METHOD TryMakeReferenceTo : BOOL
VAR_INPUT
	Target : I_Datatype;
END_VAR
VAR
	pTargetData : POINTER TO ETcVnOcrModelType;
END_VAR
IF NOT IsEquivalentTo(Target) THEN
	RETURN;
END_IF

pTargetData := Target.Address;
activeData REF= pTargetData^;
SetBaseDatatypeReference();
TryMakeReferenceTo := TRUE;
END_METHOD

PROPERTY PUBLIC Value : ETcVnOcrModelType
GET
Value := activeData;
END_GET
SET
activeData := Value;
END_SET
END_PROPERTY

END_FUNCTION_BLOCK

// ---- Datatypes/Enums/_ETcVnTimestamp.TcPOU
{attribute 'linkalways'} 
{attribute 'no_explicit_call' := 'This FB is a CLASS and must be accessed using methods or properties'}
{attribute 'enable_dynamic_creation'}
FUNCTION_BLOCK _ETcVnTimestamp EXTENDS EnumDatatypeBase
VAR
	localData : ETcVnTimestamp;
	activeData : REFERENCE TO ETcVnTimestamp;
	enumBaseDatatype : _ULINT(localData);
END_VAR

METHOD PRIVATE AddLocalEnumeration
VAR_INPUT
	Enumeration : T_MAXSTRING;
	Value : ETcVnTimestamp;
END_VAR
AddEnumeration(Enumeration, Value);
END_METHOD

PROPERTY PUBLIC Address : PVOID
GET
Address := ADR(activeData);
END_GET
END_PROPERTY

METHOD PUBLIC ClearReference
VAR_INPUT
END_VAR
activeData REF= localData;
SetBaseDatatypeReference();
END_METHOD

METHOD PUBLIC Clone : I_Datatype
VAR
    pClone : POINTER TO _ETcVnTimestamp;
END_VAR
pClone := __NEW(_ETcVnTimestamp(InitialValue := Value));
Clone := pClone^;
END_METHOD

METHOD FB_init : BOOL
VAR_INPUT
	bInitRetains : BOOL; // if TRUE, the retain variables are initialized (warm start / cold start)
	bInCopyCode : BOOL;  // if TRUE, the instance afterwards gets moved into the copy code (online change)
	InitialValue : ETcVnTimestamp;
END_VAR
localData := InitialValue;
AddBaseDatatype(enumBaseDatatype);
ClearReference();

AddLocalEnumeration('TCVN_TS_IMAGE_COMPLETED', ETcVnTimestamp.TCVN_TS_IMAGE_COMPLETED);
END_METHOD

PROPERTY PUBLIC Identifier : T_MAXSTRING
GET
Identifier := 'ETcVnTimestamp';
END_GET
END_PROPERTY

METHOD IsEnumeratorValueEqual : BOOL
VAR_INPUT
	Enumerator : I_KeyValueForwardEnumerator;
END_VAR
VAR
	storedValue : ETcVnTimestamp;
END_VAR
IF NOT Enumerator.TryGet(storedValue) THEN
	RETURN;
END_IF

IsEnumeratorValueEqual := storedValue = activeData;
END_METHOD

METHOD PUBLIC MakeReferenceTo
VAR_INPUT
	ReferenceTarget : REFERENCE TO ETcVnTimestamp;
END_VAR
activeData REF= ReferenceTarget;
SetBaseDatatypeReference();
END_METHOD

METHOD PROTECTED SetBaseDatatypeReference
VAR_INPUT
END_VAR
enumBaseDatatype.MakeReferenceTo(activeData);
END_METHOD

PROPERTY PUBLIC Size : UDINT
GET
Size := SIZEOF(activeData);
END_GET
END_PROPERTY

METHOD TryMakeReferenceTo : BOOL
VAR_INPUT
	Target : I_Datatype;
END_VAR
VAR
	pTargetData : POINTER TO ETcVnTimestamp;
END_VAR
IF NOT IsEquivalentTo(Target) THEN
	RETURN;
END_IF

pTargetData := Target.Address;
activeData REF= pTargetData^;
SetBaseDatatypeReference();
TryMakeReferenceTo := TRUE;
END_METHOD

PROPERTY PUBLIC Value : ETcVnTimestamp
GET
Value := activeData;
END_GET
SET
activeData := Value;
END_SET
END_PROPERTY

END_FUNCTION_BLOCK

// ---- Datatypes/Enums/_ETcVnOcrOptions.TcPOU
{attribute 'linkalways'} 
{attribute 'no_explicit_call' := 'This FB is a CLASS and must be accessed using methods or properties'}
{attribute 'enable_dynamic_creation'}
FUNCTION_BLOCK _ETcVnOcrOptions EXTENDS EnumDatatypeBase
VAR
	localData : ETcVnOcrOptions;
	activeData : REFERENCE TO ETcVnOcrOptions;
	enumBaseDatatype : _UDINT(localData);
END_VAR

METHOD PRIVATE AddLocalEnumeration
VAR_INPUT
	Enumeration : T_MAXSTRING;
	Value : ETcVnOcrOptions;
END_VAR
AddEnumeration(Enumeration, Value);
END_METHOD

PROPERTY PUBLIC Address : PVOID
GET
Address := ADR(activeData);
END_GET
END_PROPERTY

METHOD PUBLIC ClearReference
VAR_INPUT
END_VAR
activeData REF= localData;
SetBaseDatatypeReference();
END_METHOD

METHOD PUBLIC Clone : I_Datatype
VAR
    pClone : POINTER TO _ETcVnOcrOptions;
END_VAR
pClone := __NEW(_ETcVnOcrOptions(InitialValue := Value));
Clone := pClone^;
END_METHOD

METHOD FB_init : BOOL
VAR_INPUT
	bInitRetains : BOOL; // if TRUE, the retain variables are initialized (warm start / cold start)
	bInCopyCode : BOOL;  // if TRUE, the instance afterwards gets moved into the copy code (online change)
	InitialValue : ETcVnOcrOptions;
END_VAR
localData := InitialValue;
AddBaseDatatype(enumBaseDatatype);
ClearReference();

AddLocalEnumeration('TCVN_OO_WITHBLANKS', ETcVnOcrOptions.TCVN_OO_WITHBLANKS);
END_METHOD

PROPERTY PUBLIC Identifier : T_MAXSTRING
GET
Identifier := 'ETcVnOcrOptions';
END_GET
END_PROPERTY

METHOD IsEnumeratorValueEqual : BOOL
VAR_INPUT
	Enumerator : I_KeyValueForwardEnumerator;
END_VAR
VAR
	storedValue : ETcVnOcrOptions;
END_VAR
IF NOT Enumerator.TryGet(storedValue) THEN
	RETURN;
END_IF

IsEnumeratorValueEqual := storedValue = activeData;
END_METHOD

METHOD PUBLIC MakeReferenceTo
VAR_INPUT
	ReferenceTarget : REFERENCE TO ETcVnOcrOptions;
END_VAR
activeData REF= ReferenceTarget;
SetBaseDatatypeReference();
END_METHOD

METHOD PROTECTED SetBaseDatatypeReference
VAR_INPUT
END_VAR
enumBaseDatatype.MakeReferenceTo(activeData);
END_METHOD

PROPERTY PUBLIC Size : UDINT
GET
Size := SIZEOF(activeData);
END_GET
END_PROPERTY

METHOD TryMakeReferenceTo : BOOL
VAR_INPUT
	Target : I_Datatype;
END_VAR
VAR
	pTargetData : POINTER TO ETcVnOcrOptions;
END_VAR
IF NOT IsEquivalentTo(Target) THEN
	RETURN;
END_IF

pTargetData := Target.Address;
activeData REF= pTargetData^;
SetBaseDatatypeReference();
TryMakeReferenceTo := TRUE;
END_METHOD

PROPERTY PUBLIC Value : ETcVnOcrOptions
GET
Value := activeData;
END_GET
SET
activeData := Value;
END_SET
END_PROPERTY

END_FUNCTION_BLOCK

// ---- Datatypes/Enums/_ETcVnOrientationMethod.TcPOU
{attribute 'linkalways'} 
{attribute 'no_explicit_call' := 'This FB is a CLASS and must be accessed using methods or properties'}
{attribute 'enable_dynamic_creation'}
FUNCTION_BLOCK _ETcVnOrientationMethod EXTENDS EnumDatatypeBase
VAR
	localData : ETcVnOrientationMethod;
	activeData : REFERENCE TO ETcVnOrientationMethod;
	enumBaseDatatype : _DINT(localData);
END_VAR

METHOD PRIVATE AddLocalEnumeration
VAR_INPUT
	Enumeration : T_MAXSTRING;
	Value : ETcVnOrientationMethod;
END_VAR
AddEnumeration(Enumeration, Value);
END_METHOD

PROPERTY PUBLIC Address : PVOID
GET
Address := ADR(activeData);
END_GET
END_PROPERTY

METHOD PUBLIC ClearReference
VAR_INPUT
END_VAR
activeData REF= localData;
SetBaseDatatypeReference();
END_METHOD

METHOD PUBLIC Clone : I_Datatype
VAR
    pClone : POINTER TO _ETcVnOrientationMethod;
END_VAR
pClone := __NEW(_ETcVnOrientationMethod(InitialValue := Value));
Clone := pClone^;
END_METHOD

METHOD FB_init : BOOL
VAR_INPUT
	bInitRetains : BOOL; // if TRUE, the retain variables are initialized (warm start / cold start)
	bInCopyCode : BOOL;  // if TRUE, the instance afterwards gets moved into the copy code (online change)
	InitialValue : ETcVnOrientationMethod;
END_VAR
localData := InitialValue;
AddBaseDatatype(enumBaseDatatype);
ClearReference();

AddLocalEnumeration('TCVN_OM_PCA', ETcVnOrientationMethod.TCVN_OM_PCA);
AddLocalEnumeration('TCVN_OM_FITELLIPSE', ETcVnOrientationMethod.TCVN_OM_FITELLIPSE);
AddLocalEnumeration('TCVN_OM_MOMENTS', ETcVnOrientationMethod.TCVN_OM_MOMENTS);
AddLocalEnumeration('TCVN_OM_ENCLOSINGRECT', ETcVnOrientationMethod.TCVN_OM_ENCLOSINGRECT);
END_METHOD

PROPERTY PUBLIC Identifier : T_MAXSTRING
GET
Identifier := 'ETcVnOrientationMethod';
END_GET
END_PROPERTY

METHOD IsEnumeratorValueEqual : BOOL
VAR_INPUT
	Enumerator : I_KeyValueForwardEnumerator;
END_VAR
VAR
	storedValue : ETcVnOrientationMethod;
END_VAR
IF NOT Enumerator.TryGet(storedValue) THEN
	RETURN;
END_IF

IsEnumeratorValueEqual := storedValue = activeData;
END_METHOD

METHOD PUBLIC MakeReferenceTo
VAR_INPUT
	ReferenceTarget : REFERENCE TO ETcVnOrientationMethod;
END_VAR
activeData REF= ReferenceTarget;
SetBaseDatatypeReference();
END_METHOD

METHOD PROTECTED SetBaseDatatypeReference
VAR_INPUT
END_VAR
enumBaseDatatype.MakeReferenceTo(activeData);
END_METHOD

PROPERTY PUBLIC Size : UDINT
GET
Size := SIZEOF(activeData);
END_GET
END_PROPERTY

METHOD TryMakeReferenceTo : BOOL
VAR_INPUT
	Target : I_Datatype;
END_VAR
VAR
	pTargetData : POINTER TO ETcVnOrientationMethod;
END_VAR
IF NOT IsEquivalentTo(Target) THEN
	RETURN;
END_IF

pTargetData := Target.Address;
activeData REF= pTargetData^;
SetBaseDatatypeReference();
TryMakeReferenceTo := TRUE;
END_METHOD

PROPERTY PUBLIC Value : ETcVnOrientationMethod
GET
Value := activeData;
END_GET
SET
activeData := Value;
END_SET
END_PROPERTY

END_FUNCTION_BLOCK

// ---- Datatypes/Enums/_ETcVnPaddingMode.TcPOU
{attribute 'linkalways'} 
{attribute 'no_explicit_call' := 'This FB is a CLASS and must be accessed using methods or properties'}
{attribute 'enable_dynamic_creation'}
FUNCTION_BLOCK _ETcVnPaddingMode EXTENDS EnumDatatypeBase
VAR
	localData : ETcVnPaddingMode;
	activeData : REFERENCE TO ETcVnPaddingMode;
	enumBaseDatatype : _DINT(localData);
END_VAR

METHOD PRIVATE AddLocalEnumeration
VAR_INPUT
	Enumeration : T_MAXSTRING;
	Value : ETcVnPaddingMode;
END_VAR
AddEnumeration(Enumeration, Value);
END_METHOD

PROPERTY PUBLIC Address : PVOID
GET
Address := ADR(activeData);
END_GET
END_PROPERTY

METHOD PUBLIC ClearReference
VAR_INPUT
END_VAR
activeData REF= localData;
SetBaseDatatypeReference();
END_METHOD

METHOD PUBLIC Clone : I_Datatype
VAR
    pClone : POINTER TO _ETcVnPaddingMode;
END_VAR
pClone := __NEW(_ETcVnPaddingMode(InitialValue := Value));
Clone := pClone^;
END_METHOD

METHOD FB_init : BOOL
VAR_INPUT
	bInitRetains : BOOL; // if TRUE, the retain variables are initialized (warm start / cold start)
	bInCopyCode : BOOL;  // if TRUE, the instance afterwards gets moved into the copy code (online change)
	InitialValue : ETcVnPaddingMode;
END_VAR
localData := InitialValue;
AddBaseDatatype(enumBaseDatatype);
ClearReference();

AddLocalEnumeration('TCVN_PM_NONE', ETcVnPaddingMode.TCVN_PM_NONE);
AddLocalEnumeration('TCVN_PM_CROP_CENTER', ETcVnPaddingMode.TCVN_PM_CROP_CENTER);
AddLocalEnumeration('TCVN_PM_LETTERBOX', ETcVnPaddingMode.TCVN_PM_LETTERBOX);
END_METHOD

PROPERTY PUBLIC Identifier : T_MAXSTRING
GET
Identifier := 'ETcVnPaddingMode';
END_GET
END_PROPERTY

METHOD IsEnumeratorValueEqual : BOOL
VAR_INPUT
	Enumerator : I_KeyValueForwardEnumerator;
END_VAR
VAR
	storedValue : ETcVnPaddingMode;
END_VAR
IF NOT Enumerator.TryGet(storedValue) THEN
	RETURN;
END_IF

IsEnumeratorValueEqual := storedValue = activeData;
END_METHOD

METHOD PUBLIC MakeReferenceTo
VAR_INPUT
	ReferenceTarget : REFERENCE TO ETcVnPaddingMode;
END_VAR
activeData REF= ReferenceTarget;
SetBaseDatatypeReference();
END_METHOD

METHOD PROTECTED SetBaseDatatypeReference
VAR_INPUT
END_VAR
enumBaseDatatype.MakeReferenceTo(activeData);
END_METHOD

PROPERTY PUBLIC Size : UDINT
GET
Size := SIZEOF(activeData);
END_GET
END_PROPERTY

METHOD TryMakeReferenceTo : BOOL
VAR_INPUT
	Target : I_Datatype;
END_VAR
VAR
	pTargetData : POINTER TO ETcVnPaddingMode;
END_VAR
IF NOT IsEquivalentTo(Target) THEN
	RETURN;
END_IF

pTargetData := Target.Address;
activeData REF= pTargetData^;
SetBaseDatatypeReference();
TryMakeReferenceTo := TRUE;
END_METHOD

PROPERTY PUBLIC Value : ETcVnPaddingMode
GET
Value := activeData;
END_GET
SET
activeData := Value;
END_SET
END_PROPERTY

END_FUNCTION_BLOCK

// ---- Datatypes/Enums/_ETcVnPixelConnectivity.TcPOU
{attribute 'linkalways'} 
{attribute 'no_explicit_call' := 'This FB is a CLASS and must be accessed using methods or properties'}
{attribute 'enable_dynamic_creation'}
FUNCTION_BLOCK _ETcVnPixelConnectivity EXTENDS EnumDatatypeBase
VAR
	localData : ETcVnPixelConnectivity;
	activeData : REFERENCE TO ETcVnPixelConnectivity;
	enumBaseDatatype : _DINT(localData);
END_VAR

METHOD PRIVATE AddLocalEnumeration
VAR_INPUT
	Enumeration : T_MAXSTRING;
	Value : ETcVnPixelConnectivity;
END_VAR
AddEnumeration(Enumeration, Value);
END_METHOD

PROPERTY PUBLIC Address : PVOID
GET
Address := ADR(activeData);
END_GET
END_PROPERTY

METHOD PUBLIC ClearReference
VAR_INPUT
END_VAR
activeData REF= localData;
SetBaseDatatypeReference();
END_METHOD

METHOD PUBLIC Clone : I_Datatype
VAR
    pClone : POINTER TO _ETcVnPixelConnectivity;
END_VAR
pClone := __NEW(_ETcVnPixelConnectivity(InitialValue := Value));
Clone := pClone^;
END_METHOD

METHOD FB_init : BOOL
VAR_INPUT
	bInitRetains : BOOL; // if TRUE, the retain variables are initialized (warm start / cold start)
	bInCopyCode : BOOL;  // if TRUE, the instance afterwards gets moved into the copy code (online change)
	InitialValue : ETcVnPixelConnectivity;
END_VAR
localData := InitialValue;
AddBaseDatatype(enumBaseDatatype);
ClearReference();

AddLocalEnumeration('TCVN_PC_4', ETcVnPixelConnectivity.TCVN_PC_4);
AddLocalEnumeration('TCVN_PC_8', ETcVnPixelConnectivity.TCVN_PC_8);
END_METHOD

PROPERTY PUBLIC Identifier : T_MAXSTRING
GET
Identifier := 'ETcVnPixelConnectivity';
END_GET
END_PROPERTY

METHOD IsEnumeratorValueEqual : BOOL
VAR_INPUT
	Enumerator : I_KeyValueForwardEnumerator;
END_VAR
VAR
	storedValue : ETcVnPixelConnectivity;
END_VAR
IF NOT Enumerator.TryGet(storedValue) THEN
	RETURN;
END_IF

IsEnumeratorValueEqual := storedValue = activeData;
END_METHOD

METHOD PUBLIC MakeReferenceTo
VAR_INPUT
	ReferenceTarget : REFERENCE TO ETcVnPixelConnectivity;
END_VAR
activeData REF= ReferenceTarget;
SetBaseDatatypeReference();
END_METHOD

METHOD PROTECTED SetBaseDatatypeReference
VAR_INPUT
END_VAR
enumBaseDatatype.MakeReferenceTo(activeData);
END_METHOD

PROPERTY PUBLIC Size : UDINT
GET
Size := SIZEOF(activeData);
END_GET
END_PROPERTY

METHOD TryMakeReferenceTo : BOOL
VAR_INPUT
	Target : I_Datatype;
END_VAR
VAR
	targetAsEnum : I_EnumDatatype;
	pTargetData : POINTER TO ETcVnPixelConnectivity;
END_VAR
IF NOT Target.TryResolveAsEnumDatatype(targetAsEnum) THEN
	RETURN;
END_IF

IF targetAsEnum.Identifier <> Identifier THEN
	RETURN;
END_IF

pTargetData := Target.Address;
activeData REF= pTargetData^;
SetBaseDatatypeReference();
TryMakeReferenceTo := TRUE;
END_METHOD

PROPERTY PUBLIC Value : ETcVnPixelConnectivity
GET
Value := activeData;
END_GET
SET
activeData := Value;
END_SET
END_PROPERTY

END_FUNCTION_BLOCK

// ---- Datatypes/Enums/_ETcVnPrototypeClusterer.TcPOU
{attribute 'linkalways'} 
{attribute 'no_explicit_call' := 'This FB is a CLASS and must be accessed using methods or properties'}
{attribute 'enable_dynamic_creation'}
FUNCTION_BLOCK _ETcVnPrototypeClusterer EXTENDS EnumDatatypeBase
VAR
	localData : ETcVnPrototypeClusterer;
	activeData : REFERENCE TO ETcVnPrototypeClusterer;
	enumBaseDatatype : _UDINT(localData);
END_VAR

METHOD PRIVATE AddLocalEnumeration
VAR_INPUT
	Enumeration : T_MAXSTRING;
	Value : ETcVnPrototypeClusterer;
END_VAR
AddEnumeration(Enumeration, Value);
END_METHOD

PROPERTY PUBLIC Address : PVOID
GET
Address := ADR(activeData);
END_GET
END_PROPERTY

METHOD PUBLIC ClearReference
VAR_INPUT
END_VAR
activeData REF= localData;
SetBaseDatatypeReference();
END_METHOD

METHOD PUBLIC Clone : I_Datatype
VAR
    pClone : POINTER TO _ETcVnPrototypeClusterer;
END_VAR
pClone := __NEW(_ETcVnPrototypeClusterer(InitialValue := Value));
Clone := pClone^;
END_METHOD

METHOD FB_init : BOOL
VAR_INPUT
	bInitRetains : BOOL; // if TRUE, the retain variables are initialized (warm start / cold start)
	bInCopyCode : BOOL;  // if TRUE, the instance afterwards gets moved into the copy code (online change)
	InitialValue : ETcVnPrototypeClusterer;
END_VAR
localData := InitialValue;
AddBaseDatatype(enumBaseDatatype);
ClearReference();

AddLocalEnumeration('TCVN_PC_NOVELTY_DETECTOR', ETcVnPrototypeClusterer.TCVN_PC_NOVELTY_DETECTOR);
AddLocalEnumeration('TCVN_PC_CLUSTERER', ETcVnPrototypeClusterer.TCVN_PC_CLUSTERER);
END_METHOD

PROPERTY PUBLIC Identifier : T_MAXSTRING
GET
Identifier := 'ETcVnPrototypeClusterer';
END_GET
END_PROPERTY

METHOD IsEnumeratorValueEqual : BOOL
VAR_INPUT
	Enumerator : I_KeyValueForwardEnumerator;
END_VAR
VAR
	storedValue : ETcVnPrototypeClusterer;
END_VAR
IF NOT Enumerator.TryGet(storedValue) THEN
	RETURN;
END_IF

IsEnumeratorValueEqual := storedValue = activeData;
END_METHOD

METHOD PUBLIC MakeReferenceTo
VAR_INPUT
	ReferenceTarget : REFERENCE TO ETcVnPrototypeClusterer;
END_VAR
activeData REF= ReferenceTarget;
SetBaseDatatypeReference();
END_METHOD

METHOD PROTECTED SetBaseDatatypeReference
VAR_INPUT
END_VAR
enumBaseDatatype.MakeReferenceTo(activeData);
END_METHOD

PROPERTY PUBLIC Size : UDINT
GET
Size := SIZEOF(activeData);
END_GET
END_PROPERTY

METHOD TryMakeReferenceTo : BOOL
VAR_INPUT
	Target : I_Datatype;
END_VAR
VAR
	pTargetData : POINTER TO ETcVnPrototypeClusterer;
END_VAR
IF NOT IsEquivalentTo(Target) THEN
	RETURN;
END_IF

pTargetData := Target.Address;
activeData REF= pTargetData^;
SetBaseDatatypeReference();
TryMakeReferenceTo := TRUE;
END_METHOD

PROPERTY PUBLIC Value : ETcVnPrototypeClusterer
GET
Value := activeData;
END_GET
SET
activeData := Value;
END_SET
END_PROPERTY

END_FUNCTION_BLOCK

// ---- Datatypes/Enums/_ETcVnRectangleIntersection.TcPOU
{attribute 'linkalways'} 
{attribute 'no_explicit_call' := 'This FB is a CLASS and must be accessed using methods or properties'}
{attribute 'enable_dynamic_creation'}
FUNCTION_BLOCK _ETcVnRectangleIntersection EXTENDS EnumDatatypeBase
VAR
	localData : ETcVnRectangleIntersection;
	activeData : REFERENCE TO ETcVnRectangleIntersection;
	enumBaseDatatype : _DINT(localData);
END_VAR

METHOD PRIVATE AddLocalEnumeration
VAR_INPUT
	Enumeration : T_MAXSTRING;
	Value : ETcVnRectangleIntersection;
END_VAR
AddEnumeration(Enumeration, Value);
END_METHOD

PROPERTY PUBLIC Address : PVOID
GET
Address := ADR(activeData);
END_GET
END_PROPERTY

METHOD PUBLIC ClearReference
VAR_INPUT
END_VAR
activeData REF= localData;
SetBaseDatatypeReference();
END_METHOD

METHOD PUBLIC Clone : I_Datatype
VAR
    pClone : POINTER TO _ETcVnRectangleIntersection;
END_VAR
pClone := __NEW(_ETcVnRectangleIntersection(InitialValue := Value));
Clone := pClone^;
END_METHOD

METHOD FB_init : BOOL
VAR_INPUT
	bInitRetains : BOOL; // if TRUE, the retain variables are initialized (warm start / cold start)
	bInCopyCode : BOOL;  // if TRUE, the instance afterwards gets moved into the copy code (online change)
	InitialValue : ETcVnRectangleIntersection;
END_VAR
localData := InitialValue;
AddBaseDatatype(enumBaseDatatype);
ClearReference();

AddLocalEnumeration('TCVN_RI_NONE', ETcVnRectangleIntersection.TCVN_RI_NONE);
AddLocalEnumeration('TCVN_RI_PARTIAL', ETcVnRectangleIntersection.TCVN_RI_PARTIAL);
AddLocalEnumeration('TCVN_RI_FULL', ETcVnRectangleIntersection.TCVN_RI_FULL);
END_METHOD

PROPERTY PUBLIC Identifier : T_MAXSTRING
GET
Identifier := 'ETcVnRectangleIntersection';
END_GET
END_PROPERTY

METHOD IsEnumeratorValueEqual : BOOL
VAR_INPUT
	Enumerator : I_KeyValueForwardEnumerator;
END_VAR
VAR
	storedValue : ETcVnRectangleIntersection;
END_VAR
IF NOT Enumerator.TryGet(storedValue) THEN
	RETURN;
END_IF

IsEnumeratorValueEqual := storedValue = activeData;
END_METHOD

METHOD PUBLIC MakeReferenceTo
VAR_INPUT
	ReferenceTarget : REFERENCE TO ETcVnRectangleIntersection;
END_VAR
activeData REF= ReferenceTarget;
SetBaseDatatypeReference();
END_METHOD

METHOD PROTECTED SetBaseDatatypeReference
VAR_INPUT
END_VAR
enumBaseDatatype.MakeReferenceTo(activeData);
END_METHOD

PROPERTY PUBLIC Size : UDINT
GET
Size := SIZEOF(activeData);
END_GET
END_PROPERTY

METHOD TryMakeReferenceTo : BOOL
VAR_INPUT
	Target : I_Datatype;
END_VAR
VAR
	targetAsEnum : I_EnumDatatype;
	pTargetData : POINTER TO ETcVnRectangleIntersection;
END_VAR
IF NOT Target.TryResolveAsEnumDatatype(targetAsEnum) THEN
	RETURN;
END_IF

IF targetAsEnum.Identifier <> Identifier THEN
	RETURN;
END_IF

pTargetData := Target.Address;
activeData REF= pTargetData^;
SetBaseDatatypeReference();
TryMakeReferenceTo := TRUE;
END_METHOD

PROPERTY PUBLIC Value : ETcVnRectangleIntersection
GET
Value := activeData;
END_GET
SET
activeData := Value;
END_SET
END_PROPERTY

END_FUNCTION_BLOCK

// ---- Datatypes/Enums/_ETcVnRotationAngle.TcPOU
{attribute 'linkalways'} 
{attribute 'no_explicit_call' := 'This FB is a CLASS and must be accessed using methods or properties'}
{attribute 'enable_dynamic_creation'}
FUNCTION_BLOCK _ETcVnRotationAngle EXTENDS EnumDatatypeBase
VAR
	localData : ETcVnRotationAngle;
	activeData : REFERENCE TO ETcVnRotationAngle;
	enumBaseDatatype : _DINT(localData);
END_VAR

METHOD PRIVATE AddLocalEnumeration
VAR_INPUT
	Enumeration : T_MAXSTRING;
	Value : ETcVnRotationAngle;
END_VAR
AddEnumeration(Enumeration, Value);
END_METHOD

PROPERTY PUBLIC Address : PVOID
GET
Address := ADR(activeData);
END_GET
END_PROPERTY

METHOD PUBLIC ClearReference
VAR_INPUT
END_VAR
activeData REF= localData;
SetBaseDatatypeReference();
END_METHOD

METHOD PUBLIC Clone : I_Datatype
VAR
    pClone : POINTER TO _ETcVnRotationAngle;
END_VAR
pClone := __NEW(_ETcVnRotationAngle(InitialValue := Value));
Clone := pClone^;
END_METHOD

METHOD FB_init : BOOL
VAR_INPUT
	bInitRetains : BOOL; // if TRUE, the retain variables are initialized (warm start / cold start)
	bInCopyCode : BOOL;  // if TRUE, the instance afterwards gets moved into the copy code (online change)
	InitialValue : ETcVnRotationAngle;
END_VAR
localData := InitialValue;
AddBaseDatatype(enumBaseDatatype);
ClearReference();

AddLocalEnumeration('TCVN_RA_90_DEG', ETcVnRotationAngle.TCVN_RA_90_DEG);
AddLocalEnumeration('TCVN_RA_180_DEG', ETcVnRotationAngle.TCVN_RA_180_DEG);
AddLocalEnumeration('TCVN_RA_270_DEG', ETcVnRotationAngle.TCVN_RA_270_DEG);
END_METHOD

PROPERTY PUBLIC Identifier : T_MAXSTRING
GET
Identifier := 'ETcVnRotationAngle';
END_GET
END_PROPERTY

METHOD IsEnumeratorValueEqual : BOOL
VAR_INPUT
	Enumerator : I_KeyValueForwardEnumerator;
END_VAR
VAR
	storedValue : ETcVnRotationAngle;
END_VAR
IF NOT Enumerator.TryGet(storedValue) THEN
	RETURN;
END_IF

IsEnumeratorValueEqual := storedValue = activeData;
END_METHOD

METHOD PUBLIC MakeReferenceTo
VAR_INPUT
	ReferenceTarget : REFERENCE TO ETcVnRotationAngle;
END_VAR
activeData REF= ReferenceTarget;
SetBaseDatatypeReference();
END_METHOD

METHOD PROTECTED SetBaseDatatypeReference
VAR_INPUT
END_VAR
enumBaseDatatype.MakeReferenceTo(activeData);
END_METHOD

PROPERTY PUBLIC Size : UDINT
GET
Size := SIZEOF(activeData);
END_GET
END_PROPERTY

METHOD TryMakeReferenceTo : BOOL
VAR_INPUT
	Target : I_Datatype;
END_VAR
VAR
	targetAsEnum : I_EnumDatatype;
	pTargetData : POINTER TO ETcVnRotationAngle;
END_VAR
IF NOT Target.TryResolveAsEnumDatatype(targetAsEnum) THEN
	RETURN;
END_IF

IF targetAsEnum.Identifier <> Identifier THEN
	RETURN;
END_IF

pTargetData := Target.Address;
activeData REF= pTargetData^;
SetBaseDatatypeReference();
TryMakeReferenceTo := TRUE;
END_METHOD

PROPERTY PUBLIC Value : ETcVnRotationAngle
GET
Value := activeData;
END_GET
SET
activeData := Value;
END_SET
END_PROPERTY

END_FUNCTION_BLOCK

// ---- Datatypes/Enums/_ETcVnRTrees.TcPOU
{attribute 'linkalways'} 
{attribute 'no_explicit_call' := 'This FB is a CLASS and must be accessed using methods or properties'}
{attribute 'enable_dynamic_creation'}
FUNCTION_BLOCK _ETcVnRTrees EXTENDS EnumDatatypeBase
VAR
	localData : ETcVnRTrees;
	activeData : REFERENCE TO ETcVnRTrees;
	enumBaseDatatype : _UDINT(localData);
END_VAR

METHOD PRIVATE AddLocalEnumeration
VAR_INPUT
	Enumeration : T_MAXSTRING;
	Value : ETcVnRTrees;
END_VAR
AddEnumeration(Enumeration, Value);
END_METHOD

PROPERTY PUBLIC Address : PVOID
GET
Address := ADR(activeData);
END_GET
END_PROPERTY

METHOD PUBLIC ClearReference
VAR_INPUT
END_VAR
activeData REF= localData;
SetBaseDatatypeReference();
END_METHOD

METHOD PUBLIC Clone : I_Datatype
VAR
    pClone : POINTER TO _ETcVnRTrees;
END_VAR
pClone := __NEW(_ETcVnRTrees(InitialValue := Value));
Clone := pClone^;
END_METHOD

METHOD FB_init : BOOL
VAR_INPUT
	bInitRetains : BOOL; // if TRUE, the retain variables are initialized (warm start / cold start)
	bInCopyCode : BOOL;  // if TRUE, the instance afterwards gets moved into the copy code (online change)
	InitialValue : ETcVnRTrees;
END_VAR
localData := InitialValue;
AddBaseDatatype(enumBaseDatatype);
ClearReference();

AddLocalEnumeration('TCVN_RT_CLASSIFIER', ETcVnRTrees.TCVN_RT_CLASSIFIER);
AddLocalEnumeration('TCVN_RT_REGRESSOR', ETcVnRTrees.TCVN_RT_REGRESSOR);
END_METHOD

PROPERTY PUBLIC Identifier : T_MAXSTRING
GET
Identifier := 'ETcVnRTrees';
END_GET
END_PROPERTY

METHOD IsEnumeratorValueEqual : BOOL
VAR_INPUT
	Enumerator : I_KeyValueForwardEnumerator;
END_VAR
VAR
	storedValue : ETcVnRTrees;
END_VAR
IF NOT Enumerator.TryGet(storedValue) THEN
	RETURN;
END_IF

IsEnumeratorValueEqual := storedValue = activeData;
END_METHOD

METHOD PUBLIC MakeReferenceTo
VAR_INPUT
	ReferenceTarget : REFERENCE TO ETcVnRTrees;
END_VAR
activeData REF= ReferenceTarget;
SetBaseDatatypeReference();
END_METHOD

METHOD PROTECTED SetBaseDatatypeReference
VAR_INPUT
END_VAR
enumBaseDatatype.MakeReferenceTo(activeData);
END_METHOD

PROPERTY PUBLIC Size : UDINT
GET
Size := SIZEOF(activeData);
END_GET
END_PROPERTY

METHOD TryMakeReferenceTo : BOOL
VAR_INPUT
	Target : I_Datatype;
END_VAR
VAR
	pTargetData : POINTER TO ETcVnRTrees;
END_VAR
IF NOT IsEquivalentTo(Target) THEN
	RETURN;
END_IF

pTargetData := Target.Address;
activeData REF= pTargetData^;
SetBaseDatatypeReference();
TryMakeReferenceTo := TRUE;
END_METHOD

PROPERTY PUBLIC Value : ETcVnRTrees
GET
Value := activeData;
END_GET
SET
activeData := Value;
END_SET
END_PROPERTY

END_FUNCTION_BLOCK

// ---- Datatypes/Enums/_ETcVnSignedNormalization.TcPOU
{attribute 'linkalways'} 
{attribute 'no_explicit_call' := 'This FB is a CLASS and must be accessed using methods or properties'}
{attribute 'enable_dynamic_creation'}
FUNCTION_BLOCK _ETcVnSignedNormalization EXTENDS EnumDatatypeBase
VAR
	localData : ETcVnSignedNormalization;
	activeData : REFERENCE TO ETcVnSignedNormalization;
	enumBaseDatatype : _INT(localData);
END_VAR

METHOD PRIVATE AddLocalEnumeration
VAR_INPUT
	Enumeration : T_MAXSTRING;
	Value : ETcVnSignedNormalization;
END_VAR
AddEnumeration(Enumeration, Value);
END_METHOD

PROPERTY PUBLIC Address : PVOID
GET
Address := ADR(activeData);
END_GET
END_PROPERTY

METHOD PUBLIC ClearReference
VAR_INPUT
END_VAR
activeData REF= localData;
SetBaseDatatypeReference();
END_METHOD

METHOD PUBLIC Clone : I_Datatype
VAR
    pClone : POINTER TO _ETcVnSignedNormalization;
END_VAR
pClone := __NEW(_ETcVnSignedNormalization(InitialValue := Value));
Clone := pClone^;
END_METHOD

METHOD FB_init : BOOL
VAR_INPUT
	bInitRetains : BOOL; // if TRUE, the retain variables are initialized (warm start / cold start)
	bInCopyCode : BOOL;  // if TRUE, the instance afterwards gets moved into the copy code (online change)
	InitialValue : ETcVnSignedNormalization;
END_VAR
localData := InitialValue;
AddBaseDatatype(enumBaseDatatype);
ClearReference();

AddLocalEnumeration('TCVN_SN_FIX_ZERO', ETcVnSignedNormalization.TCVN_SN_FIX_ZERO);
AddLocalEnumeration('TCVN_SN_FULL_SCALE', ETcVnSignedNormalization.TCVN_SN_FULL_SCALE);
END_METHOD

PROPERTY PUBLIC Identifier : T_MAXSTRING
GET
Identifier := 'ETcVnSignedNormalization';
END_GET
END_PROPERTY

METHOD IsEnumeratorValueEqual : BOOL
VAR_INPUT
	Enumerator : I_KeyValueForwardEnumerator;
END_VAR
VAR
	storedValue : ETcVnSignedNormalization;
END_VAR
IF NOT Enumerator.TryGet(storedValue) THEN
	RETURN;
END_IF

IsEnumeratorValueEqual := storedValue = activeData;
END_METHOD

METHOD PUBLIC MakeReferenceTo
VAR_INPUT
	ReferenceTarget : REFERENCE TO ETcVnSignedNormalization;
END_VAR
activeData REF= ReferenceTarget;
SetBaseDatatypeReference();
END_METHOD

METHOD PROTECTED SetBaseDatatypeReference
VAR_INPUT
END_VAR
enumBaseDatatype.MakeReferenceTo(activeData);
END_METHOD

PROPERTY PUBLIC Size : UDINT
GET
Size := SIZEOF(activeData);
END_GET
END_PROPERTY

METHOD TryMakeReferenceTo : BOOL
VAR_INPUT
	Target : I_Datatype;
END_VAR
VAR
	pTargetData : POINTER TO ETcVnSignedNormalization;
END_VAR
IF NOT IsEquivalentTo(Target) THEN
	RETURN;
END_IF

pTargetData := Target.Address;
activeData REF= pTargetData^;
SetBaseDatatypeReference();
TryMakeReferenceTo := TRUE;
END_METHOD

PROPERTY PUBLIC Value : ETcVnSignedNormalization
GET
Value := activeData;
END_GET
SET
activeData := Value;
END_SET
END_PROPERTY

END_FUNCTION_BLOCK

// ---- Datatypes/Enums/_ETcVnSolvePnPMethod.TcPOU
{attribute 'linkalways'} 
{attribute 'no_explicit_call' := 'This FB is a CLASS and must be accessed using methods or properties'}
{attribute 'enable_dynamic_creation'}
FUNCTION_BLOCK _ETcVnSolvePnPMethod EXTENDS EnumDatatypeBase
VAR
	localData : ETcVnSolvePnPMethod;
	activeData : REFERENCE TO ETcVnSolvePnPMethod;
	enumBaseDatatype : _DINT(localData);
END_VAR

METHOD PRIVATE AddLocalEnumeration
VAR_INPUT
	Enumeration : T_MAXSTRING;
	Value : ETcVnSolvePnPMethod;
END_VAR
AddEnumeration(Enumeration, Value);
END_METHOD

PROPERTY PUBLIC Address : PVOID
GET
Address := ADR(activeData);
END_GET
END_PROPERTY

METHOD PUBLIC ClearReference
VAR_INPUT
END_VAR
activeData REF= localData;
SetBaseDatatypeReference();
END_METHOD

METHOD PUBLIC Clone : I_Datatype
VAR
    pClone : POINTER TO _ETcVnSolvePnPMethod;
END_VAR
pClone := __NEW(_ETcVnSolvePnPMethod(InitialValue := Value));
Clone := pClone^;
END_METHOD

METHOD FB_init : BOOL
VAR_INPUT
	bInitRetains : BOOL; // if TRUE, the retain variables are initialized (warm start / cold start)
	bInCopyCode : BOOL;  // if TRUE, the instance afterwards gets moved into the copy code (online change)
	InitialValue : ETcVnSolvePnPMethod;
END_VAR
localData := InitialValue;
AddBaseDatatype(enumBaseDatatype);
ClearReference();

AddLocalEnumeration('TCVN_SPM_ITERATIVE', ETcVnSolvePnPMethod.TCVN_SPM_ITERATIVE);
AddLocalEnumeration('TCVN_SPM_EPNP', ETcVnSolvePnPMethod.TCVN_SPM_EPNP);
AddLocalEnumeration('TCVN_SPM_P3P', ETcVnSolvePnPMethod.TCVN_SPM_P3P);
AddLocalEnumeration('TCVN_SPM_AP3P', ETcVnSolvePnPMethod.TCVN_SPM_AP3P);
AddLocalEnumeration('TCVN_SPM_IPPE', ETcVnSolvePnPMethod.TCVN_SPM_IPPE);
AddLocalEnumeration('TCVN_SPM_IPPE_SQUARE', ETcVnSolvePnPMethod.TCVN_SPM_IPPE_SQUARE);
AddLocalEnumeration('TCVN_SPM_SQPNP', ETcVnSolvePnPMethod.TCVN_SPM_SQPNP);
END_METHOD

PROPERTY PUBLIC Identifier : T_MAXSTRING
GET
Identifier := 'ETcVnSolvePnPMethod';
END_GET
END_PROPERTY

METHOD IsEnumeratorValueEqual : BOOL
VAR_INPUT
	Enumerator : I_KeyValueForwardEnumerator;
END_VAR
VAR
	storedValue : ETcVnSolvePnPMethod;
END_VAR
IF NOT Enumerator.TryGet(storedValue) THEN
	RETURN;
END_IF

IsEnumeratorValueEqual := storedValue = activeData;
END_METHOD

METHOD PUBLIC MakeReferenceTo
VAR_INPUT
	ReferenceTarget : REFERENCE TO ETcVnSolvePnPMethod;
END_VAR
activeData REF= ReferenceTarget;
SetBaseDatatypeReference();
END_METHOD

METHOD PROTECTED SetBaseDatatypeReference
VAR_INPUT
END_VAR
enumBaseDatatype.MakeReferenceTo(activeData);
END_METHOD

PROPERTY PUBLIC Size : UDINT
GET
Size := SIZEOF(activeData);
END_GET
END_PROPERTY

METHOD TryMakeReferenceTo : BOOL
VAR_INPUT
	Target : I_Datatype;
END_VAR
VAR
	pTargetData : POINTER TO ETcVnSolvePnPMethod;
END_VAR
IF NOT IsEquivalentTo(Target) THEN
	RETURN;
END_IF

pTargetData := Target.Address;
activeData REF= pTargetData^;
SetBaseDatatypeReference();
TryMakeReferenceTo := TRUE;
END_METHOD

PROPERTY PUBLIC Value : ETcVnSolvePnPMethod
GET
Value := activeData;
END_GET
SET
activeData := Value;
END_SET
END_PROPERTY

END_FUNCTION_BLOCK

// ---- Datatypes/Enums/_ETcVnSta.TcPOU
{attribute 'linkalways'} 
{attribute 'no_explicit_call' := 'This FB is a CLASS and must be accessed using methods or properties'}
{attribute 'enable_dynamic_creation'}
FUNCTION_BLOCK _ETcVnSta EXTENDS EnumDatatypeBase
VAR
	localData : ETcVnSta;
	activeData : REFERENCE TO ETcVnSta;
	enumBaseDatatype : _UDINT(localData);
END_VAR

METHOD PRIVATE AddLocalEnumeration
VAR_INPUT
	Enumeration : T_MAXSTRING;
	Value : ETcVnSta;
END_VAR
AddEnumeration(Enumeration, Value);
END_METHOD

PROPERTY PUBLIC Address : PVOID
GET
Address := ADR(activeData);
END_GET
END_PROPERTY

METHOD PUBLIC ClearReference
VAR_INPUT
END_VAR
activeData REF= localData;
SetBaseDatatypeReference();
END_METHOD

METHOD PUBLIC Clone : I_Datatype
VAR
    pClone : POINTER TO _ETcVnSta;
END_VAR
pClone := __NEW(_ETcVnSta(InitialValue := Value));
Clone := pClone^;
END_METHOD

METHOD FB_init : BOOL
VAR_INPUT
	bInitRetains : BOOL; // if TRUE, the retain variables are initialized (warm start / cold start)
	bInCopyCode : BOOL;  // if TRUE, the instance afterwards gets moved into the copy code (online change)
	InitialValue : ETcVnSta;
END_VAR
localData := InitialValue;
AddBaseDatatype(enumBaseDatatype);
ClearReference();

AddLocalEnumeration('TCVN_STA_CLASSIFIER', ETcVnSta.TCVN_STA_CLASSIFIER);
AddLocalEnumeration('TCVN_STA_NOVELTY_DETECTOR', ETcVnSta.TCVN_STA_NOVELTY_DETECTOR);
AddLocalEnumeration('TCVN_STA_REGRESSOR', ETcVnSta.TCVN_STA_REGRESSOR);
AddLocalEnumeration('TCVN_STA_CLUSTERER', ETcVnSta.TCVN_STA_CLUSTERER);
END_METHOD

PROPERTY PUBLIC Identifier : T_MAXSTRING
GET
Identifier := 'ETcVnSta';
END_GET
END_PROPERTY

METHOD IsEnumeratorValueEqual : BOOL
VAR_INPUT
	Enumerator : I_KeyValueForwardEnumerator;
END_VAR
VAR
	storedValue : ETcVnSta;
END_VAR
IF NOT Enumerator.TryGet(storedValue) THEN
	RETURN;
END_IF

IsEnumeratorValueEqual := storedValue = activeData;
END_METHOD

METHOD PUBLIC MakeReferenceTo
VAR_INPUT
	ReferenceTarget : REFERENCE TO ETcVnSta;
END_VAR
activeData REF= ReferenceTarget;
SetBaseDatatypeReference();
END_METHOD

METHOD PROTECTED SetBaseDatatypeReference
VAR_INPUT
END_VAR
enumBaseDatatype.MakeReferenceTo(activeData);
END_METHOD

PROPERTY PUBLIC Size : UDINT
GET
Size := SIZEOF(activeData);
END_GET
END_PROPERTY

METHOD TryMakeReferenceTo : BOOL
VAR_INPUT
	Target : I_Datatype;
END_VAR
VAR
	pTargetData : POINTER TO ETcVnSta;
END_VAR
IF NOT IsEquivalentTo(Target) THEN
	RETURN;
END_IF

pTargetData := Target.Address;
activeData REF= pTargetData^;
SetBaseDatatypeReference();
TryMakeReferenceTo := TRUE;
END_METHOD

PROPERTY PUBLIC Value : ETcVnSta
GET
Value := activeData;
END_GET
SET
activeData := Value;
END_SET
END_PROPERTY

END_FUNCTION_BLOCK

// ---- Datatypes/Enums/_ETcVnStructuringElementShape.TcPOU
{attribute 'linkalways'} 
{attribute 'no_explicit_call' := 'This FB is a CLASS and must be accessed using methods or properties'}
{attribute 'enable_dynamic_creation'}
FUNCTION_BLOCK _ETcVnStructuringElementShape EXTENDS EnumDatatypeBase
VAR
	localData : ETcVnStructuringElementShape;
	activeData : REFERENCE TO ETcVnStructuringElementShape;
	enumBaseDatatype : _DINT(localData);
END_VAR

METHOD PRIVATE AddLocalEnumeration
VAR_INPUT
	Enumeration : T_MAXSTRING;
	Value : ETcVnStructuringElementShape;
END_VAR
AddEnumeration(Enumeration, Value);
END_METHOD

PROPERTY PUBLIC Address : PVOID
GET
Address := ADR(activeData);
END_GET
END_PROPERTY

METHOD PUBLIC ClearReference
VAR_INPUT
END_VAR
activeData REF= localData;
SetBaseDatatypeReference();
END_METHOD

METHOD PUBLIC Clone : I_Datatype
VAR
    pClone : POINTER TO _ETcVnStructuringElementShape;
END_VAR
pClone := __NEW(_ETcVnStructuringElementShape(InitialValue := Value));
Clone := pClone^;
END_METHOD

METHOD FB_init : BOOL
VAR_INPUT
	bInitRetains : BOOL; // if TRUE, the retain variables are initialized (warm start / cold start)
	bInCopyCode : BOOL;  // if TRUE, the instance afterwards gets moved into the copy code (online change)
	InitialValue : ETcVnStructuringElementShape;
END_VAR
localData := InitialValue;
AddBaseDatatype(enumBaseDatatype);
ClearReference();

AddLocalEnumeration('TCVN_SES_RECTANGLE', ETcVnStructuringElementShape.TCVN_SES_RECTANGLE);
AddLocalEnumeration('TCVN_SES_CROSS', ETcVnStructuringElementShape.TCVN_SES_CROSS);
AddLocalEnumeration('TCVN_SES_ELLIPSE', ETcVnStructuringElementShape.TCVN_SES_ELLIPSE);
END_METHOD

PROPERTY PUBLIC Identifier : T_MAXSTRING
GET
Identifier := 'ETcVnStructuringElementShape';
END_GET
END_PROPERTY

METHOD IsEnumeratorValueEqual : BOOL
VAR_INPUT
	Enumerator : I_KeyValueForwardEnumerator;
END_VAR
VAR
	storedValue : ETcVnStructuringElementShape;
END_VAR
IF NOT Enumerator.TryGet(storedValue) THEN
	RETURN;
END_IF

IsEnumeratorValueEqual := storedValue = activeData;
END_METHOD

METHOD PUBLIC MakeReferenceTo
VAR_INPUT
	ReferenceTarget : REFERENCE TO ETcVnStructuringElementShape;
END_VAR
activeData REF= ReferenceTarget;
SetBaseDatatypeReference();
END_METHOD

METHOD PROTECTED SetBaseDatatypeReference
VAR_INPUT
END_VAR
enumBaseDatatype.MakeReferenceTo(activeData);
END_METHOD

PROPERTY PUBLIC Size : UDINT
GET
Size := SIZEOF(activeData);
END_GET
END_PROPERTY

METHOD TryMakeReferenceTo : BOOL
VAR_INPUT
	Target : I_Datatype;
END_VAR
VAR
	targetAsEnum : I_EnumDatatype;
	pTargetData : POINTER TO ETcVnStructuringElementShape;
END_VAR
IF NOT Target.TryResolveAsEnumDatatype(targetAsEnum) THEN
	RETURN;
END_IF

IF targetAsEnum.Identifier <> Identifier THEN
	RETURN;
END_IF

pTargetData := Target.Address;
activeData REF= pTargetData^;
SetBaseDatatypeReference();
TryMakeReferenceTo := TRUE;
END_METHOD

PROPERTY PUBLIC Value : ETcVnStructuringElementShape
GET
Value := activeData;
END_GET
SET
activeData := Value;
END_SET
END_PROPERTY

END_FUNCTION_BLOCK

// ---- Datatypes/Enums/_ETcVnSvm.TcPOU
{attribute 'linkalways'} 
{attribute 'no_explicit_call' := 'This FB is a CLASS and must be accessed using methods or properties'}
{attribute 'enable_dynamic_creation'}
FUNCTION_BLOCK _ETcVnSvm EXTENDS EnumDatatypeBase
VAR
	localData : ETcVnSvm;
	activeData : REFERENCE TO ETcVnSvm;
	enumBaseDatatype : _UDINT(localData);
END_VAR

METHOD PRIVATE AddLocalEnumeration
VAR_INPUT
	Enumeration : T_MAXSTRING;
	Value : ETcVnSvm;
END_VAR
AddEnumeration(Enumeration, Value);
END_METHOD

PROPERTY PUBLIC Address : PVOID
GET
Address := ADR(activeData);
END_GET
END_PROPERTY

METHOD PUBLIC ClearReference
VAR_INPUT
END_VAR
activeData REF= localData;
SetBaseDatatypeReference();
END_METHOD

METHOD PUBLIC Clone : I_Datatype
VAR
    pClone : POINTER TO _ETcVnSvm;
END_VAR
pClone := __NEW(_ETcVnSvm(InitialValue := Value));
Clone := pClone^;
END_METHOD

METHOD FB_init : BOOL
VAR_INPUT
	bInitRetains : BOOL; // if TRUE, the retain variables are initialized (warm start / cold start)
	bInCopyCode : BOOL;  // if TRUE, the instance afterwards gets moved into the copy code (online change)
	InitialValue : ETcVnSvm;
END_VAR
localData := InitialValue;
AddBaseDatatype(enumBaseDatatype);
ClearReference();

AddLocalEnumeration('TCVN_SVM_C_CLASSIFIER', ETcVnSvm.TCVN_SVM_C_CLASSIFIER);
AddLocalEnumeration('TCVN_SVM_NU_CLASSIFIER', ETcVnSvm.TCVN_SVM_NU_CLASSIFIER);
AddLocalEnumeration('TCVN_SVM_NOVELTY_DETECTOR', ETcVnSvm.TCVN_SVM_NOVELTY_DETECTOR);
AddLocalEnumeration('TCVN_SVM_EPS_REGRESSOR', ETcVnSvm.TCVN_SVM_EPS_REGRESSOR);
AddLocalEnumeration('TCVN_SVM_NU_REGRESSOR', ETcVnSvm.TCVN_SVM_NU_REGRESSOR);
END_METHOD

PROPERTY PUBLIC Identifier : T_MAXSTRING
GET
Identifier := 'ETcVnSvm';
END_GET
END_PROPERTY

METHOD IsEnumeratorValueEqual : BOOL
VAR_INPUT
	Enumerator : I_KeyValueForwardEnumerator;
END_VAR
VAR
	storedValue : ETcVnSvm;
END_VAR
IF NOT Enumerator.TryGet(storedValue) THEN
	RETURN;
END_IF

IsEnumeratorValueEqual := storedValue = activeData;
END_METHOD

METHOD PUBLIC MakeReferenceTo
VAR_INPUT
	ReferenceTarget : REFERENCE TO ETcVnSvm;
END_VAR
activeData REF= ReferenceTarget;
SetBaseDatatypeReference();
END_METHOD

METHOD PROTECTED SetBaseDatatypeReference
VAR_INPUT
END_VAR
enumBaseDatatype.MakeReferenceTo(activeData);
END_METHOD

PROPERTY PUBLIC Size : UDINT
GET
Size := SIZEOF(activeData);
END_GET
END_PROPERTY

METHOD TryMakeReferenceTo : BOOL
VAR_INPUT
	Target : I_Datatype;
END_VAR
VAR
	pTargetData : POINTER TO ETcVnSvm;
END_VAR
IF NOT IsEquivalentTo(Target) THEN
	RETURN;
END_IF

pTargetData := Target.Address;
activeData REF= pTargetData^;
SetBaseDatatypeReference();
TryMakeReferenceTo := TRUE;
END_METHOD

PROPERTY PUBLIC Value : ETcVnSvm
GET
Value := activeData;
END_GET
SET
activeData := Value;
END_SET
END_PROPERTY

END_FUNCTION_BLOCK

// ---- Datatypes/Enums/_ETcVnSvmKernelType.TcPOU
{attribute 'linkalways'} 
{attribute 'no_explicit_call' := 'This FB is a CLASS and must be accessed using methods or properties'}
{attribute 'enable_dynamic_creation'}
FUNCTION_BLOCK _ETcVnSvmKernelType EXTENDS EnumDatatypeBase
VAR
	localData : ETcVnSvmKernelType;
	activeData : REFERENCE TO ETcVnSvmKernelType;
	enumBaseDatatype : _DINT(localData);
END_VAR

METHOD PRIVATE AddLocalEnumeration
VAR_INPUT
	Enumeration : T_MAXSTRING;
	Value : ETcVnSvmKernelType;
END_VAR
AddEnumeration(Enumeration, Value);
END_METHOD

PROPERTY PUBLIC Address : PVOID
GET
Address := ADR(activeData);
END_GET
END_PROPERTY

METHOD PUBLIC ClearReference
VAR_INPUT
END_VAR
activeData REF= localData;
SetBaseDatatypeReference();
END_METHOD

METHOD PUBLIC Clone : I_Datatype
VAR
    pClone : POINTER TO _ETcVnSvmKernelType;
END_VAR
pClone := __NEW(_ETcVnSvmKernelType(InitialValue := Value));
Clone := pClone^;
END_METHOD

METHOD FB_init : BOOL
VAR_INPUT
	bInitRetains : BOOL; // if TRUE, the retain variables are initialized (warm start / cold start)
	bInCopyCode : BOOL;  // if TRUE, the instance afterwards gets moved into the copy code (online change)
	InitialValue : ETcVnSvmKernelType;
END_VAR
localData := InitialValue;
AddBaseDatatype(enumBaseDatatype);
ClearReference();

AddLocalEnumeration('TCVN_SKT_LINEAR', ETcVnSvmKernelType.TCVN_SKT_LINEAR);
AddLocalEnumeration('TCVN_SKT_POLY', ETcVnSvmKernelType.TCVN_SKT_POLY);
AddLocalEnumeration('TCVN_SKT_RBF', ETcVnSvmKernelType.TCVN_SKT_RBF);
AddLocalEnumeration('TCVN_SKT_SIGMOID', ETcVnSvmKernelType.TCVN_SKT_SIGMOID);
AddLocalEnumeration('TCVN_SKT_CHI2', ETcVnSvmKernelType.TCVN_SKT_CHI2);
AddLocalEnumeration('TCVN_SKT_INTER', ETcVnSvmKernelType.TCVN_SKT_INTER);
END_METHOD

PROPERTY PUBLIC Identifier : T_MAXSTRING
GET
Identifier := 'ETcVnSvmKernelType';
END_GET
END_PROPERTY

METHOD IsEnumeratorValueEqual : BOOL
VAR_INPUT
	Enumerator : I_KeyValueForwardEnumerator;
END_VAR
VAR
	storedValue : ETcVnSvmKernelType;
END_VAR
IF NOT Enumerator.TryGet(storedValue) THEN
	RETURN;
END_IF

IsEnumeratorValueEqual := storedValue = activeData;
END_METHOD

METHOD PUBLIC MakeReferenceTo
VAR_INPUT
	ReferenceTarget : REFERENCE TO ETcVnSvmKernelType;
END_VAR
activeData REF= ReferenceTarget;
SetBaseDatatypeReference();
END_METHOD

METHOD PROTECTED SetBaseDatatypeReference
VAR_INPUT
END_VAR
enumBaseDatatype.MakeReferenceTo(activeData);
END_METHOD

PROPERTY PUBLIC Size : UDINT
GET
Size := SIZEOF(activeData);
END_GET
END_PROPERTY

METHOD TryMakeReferenceTo : BOOL
VAR_INPUT
	Target : I_Datatype;
END_VAR
VAR
	pTargetData : POINTER TO ETcVnSvmKernelType;
END_VAR
IF NOT IsEquivalentTo(Target) THEN
	RETURN;
END_IF

pTargetData := Target.Address;
activeData REF= pTargetData^;
SetBaseDatatypeReference();
TryMakeReferenceTo := TRUE;
END_METHOD

PROPERTY PUBLIC Value : ETcVnSvmKernelType
GET
Value := activeData;
END_GET
SET
activeData := Value;
END_SET
END_PROPERTY

END_FUNCTION_BLOCK

// ---- Datatypes/Enums/_ETcVnSvmSgdClassifierMarginType.TcPOU
{attribute 'linkalways'} 
{attribute 'no_explicit_call' := 'This FB is a CLASS and must be accessed using methods or properties'}
{attribute 'enable_dynamic_creation'}
FUNCTION_BLOCK _ETcVnSvmSgdClassifierMarginType EXTENDS EnumDatatypeBase
VAR
	localData : ETcVnSvmSgdClassifierMarginType;
	activeData : REFERENCE TO ETcVnSvmSgdClassifierMarginType;
	enumBaseDatatype : _DINT(localData);
END_VAR

METHOD PRIVATE AddLocalEnumeration
VAR_INPUT
	Enumeration : T_MAXSTRING;
	Value : ETcVnSvmSgdClassifierMarginType;
END_VAR
AddEnumeration(Enumeration, Value);
END_METHOD

PROPERTY PUBLIC Address : PVOID
GET
Address := ADR(activeData);
END_GET
END_PROPERTY

METHOD PUBLIC ClearReference
VAR_INPUT
END_VAR
activeData REF= localData;
SetBaseDatatypeReference();
END_METHOD

METHOD PUBLIC Clone : I_Datatype
VAR
    pClone : POINTER TO _ETcVnSvmSgdClassifierMarginType;
END_VAR
pClone := __NEW(_ETcVnSvmSgdClassifierMarginType(InitialValue := Value));
Clone := pClone^;
END_METHOD

METHOD FB_init : BOOL
VAR_INPUT
	bInitRetains : BOOL; // if TRUE, the retain variables are initialized (warm start / cold start)
	bInCopyCode : BOOL;  // if TRUE, the instance afterwards gets moved into the copy code (online change)
	InitialValue : ETcVnSvmSgdClassifierMarginType;
END_VAR
localData := InitialValue;
AddBaseDatatype(enumBaseDatatype);
ClearReference();

AddLocalEnumeration('TCVN_SSCMT_SOFT_MARGIN', ETcVnSvmSgdClassifierMarginType.TCVN_SSCMT_SOFT_MARGIN);
AddLocalEnumeration('TCVN_SSCMT_HARD_MARGIN', ETcVnSvmSgdClassifierMarginType.TCVN_SSCMT_HARD_MARGIN);
END_METHOD

PROPERTY PUBLIC Identifier : T_MAXSTRING
GET
Identifier := 'ETcVnSvmSgdClassifierMarginType';
END_GET
END_PROPERTY

METHOD IsEnumeratorValueEqual : BOOL
VAR_INPUT
	Enumerator : I_KeyValueForwardEnumerator;
END_VAR
VAR
	storedValue : ETcVnSvmSgdClassifierMarginType;
END_VAR
IF NOT Enumerator.TryGet(storedValue) THEN
	RETURN;
END_IF

IsEnumeratorValueEqual := storedValue = activeData;
END_METHOD

METHOD PUBLIC MakeReferenceTo
VAR_INPUT
	ReferenceTarget : REFERENCE TO ETcVnSvmSgdClassifierMarginType;
END_VAR
activeData REF= ReferenceTarget;
SetBaseDatatypeReference();
END_METHOD

METHOD PROTECTED SetBaseDatatypeReference
VAR_INPUT
END_VAR
enumBaseDatatype.MakeReferenceTo(activeData);
END_METHOD

PROPERTY PUBLIC Size : UDINT
GET
Size := SIZEOF(activeData);
END_GET
END_PROPERTY

METHOD TryMakeReferenceTo : BOOL
VAR_INPUT
	Target : I_Datatype;
END_VAR
VAR
	targetAsEnum : I_EnumDatatype;
	pTargetData : POINTER TO ETcVnSvmSgdClassifierMarginType;
END_VAR
IF NOT Target.TryResolveAsEnumDatatype(targetAsEnum) THEN
	RETURN;
END_IF

IF targetAsEnum.Identifier <> Identifier THEN
	RETURN;
END_IF

pTargetData := Target.Address;
activeData REF= pTargetData^;
SetBaseDatatypeReference();
TryMakeReferenceTo := TRUE;
END_METHOD

PROPERTY PUBLIC Value : ETcVnSvmSgdClassifierMarginType
GET
Value := activeData;
END_GET
SET
activeData := Value;
END_SET
END_PROPERTY

END_FUNCTION_BLOCK

// ---- Datatypes/Enums/_ETcVnSvmSgdClassifierType.TcPOU
{attribute 'linkalways'} 
{attribute 'no_explicit_call' := 'This FB is a CLASS and must be accessed using methods or properties'}
{attribute 'enable_dynamic_creation'}
FUNCTION_BLOCK _ETcVnSvmSgdClassifierType EXTENDS EnumDatatypeBase
VAR
	localData : ETcVnSvmSgdClassifierType;
	activeData : REFERENCE TO ETcVnSvmSgdClassifierType;
	enumBaseDatatype : _DINT(localData);
END_VAR

METHOD PRIVATE AddLocalEnumeration
VAR_INPUT
	Enumeration : T_MAXSTRING;
	Value : ETcVnSvmSgdClassifierType;
END_VAR
AddEnumeration(Enumeration, Value);
END_METHOD

PROPERTY PUBLIC Address : PVOID
GET
Address := ADR(activeData);
END_GET
END_PROPERTY

METHOD PUBLIC ClearReference
VAR_INPUT
END_VAR
activeData REF= localData;
SetBaseDatatypeReference();
END_METHOD

METHOD PUBLIC Clone : I_Datatype
VAR
    pClone : POINTER TO _ETcVnSvmSgdClassifierType;
END_VAR
pClone := __NEW(_ETcVnSvmSgdClassifierType(InitialValue := Value));
Clone := pClone^;
END_METHOD

METHOD FB_init : BOOL
VAR_INPUT
	bInitRetains : BOOL; // if TRUE, the retain variables are initialized (warm start / cold start)
	bInCopyCode : BOOL;  // if TRUE, the instance afterwards gets moved into the copy code (online change)
	InitialValue : ETcVnSvmSgdClassifierType;
END_VAR
localData := InitialValue;
AddBaseDatatype(enumBaseDatatype);
ClearReference();

AddLocalEnumeration('TCVN_SSCT_SGD', ETcVnSvmSgdClassifierType.TCVN_SSCT_SGD);
AddLocalEnumeration('TCVN_SSCT_ASGD', ETcVnSvmSgdClassifierType.TCVN_SSCT_ASGD);
END_METHOD

PROPERTY PUBLIC Identifier : T_MAXSTRING
GET
Identifier := 'ETcVnSvmSgdClassifierType';
END_GET
END_PROPERTY

METHOD IsEnumeratorValueEqual : BOOL
VAR_INPUT
	Enumerator : I_KeyValueForwardEnumerator;
END_VAR
VAR
	storedValue : ETcVnSvmSgdClassifierType;
END_VAR
IF NOT Enumerator.TryGet(storedValue) THEN
	RETURN;
END_IF

IsEnumeratorValueEqual := storedValue = activeData;
END_METHOD

METHOD PUBLIC MakeReferenceTo
VAR_INPUT
	ReferenceTarget : REFERENCE TO ETcVnSvmSgdClassifierType;
END_VAR
activeData REF= ReferenceTarget;
SetBaseDatatypeReference();
END_METHOD

METHOD PROTECTED SetBaseDatatypeReference
VAR_INPUT
END_VAR
enumBaseDatatype.MakeReferenceTo(activeData);
END_METHOD

PROPERTY PUBLIC Size : UDINT
GET
Size := SIZEOF(activeData);
END_GET
END_PROPERTY

METHOD TryMakeReferenceTo : BOOL
VAR_INPUT
	Target : I_Datatype;
END_VAR
VAR
	pTargetData : POINTER TO ETcVnSvmSgdClassifierType;
END_VAR
IF NOT IsEquivalentTo(Target) THEN
	RETURN;
END_IF

pTargetData := Target.Address;
activeData REF= pTargetData^;
SetBaseDatatypeReference();
TryMakeReferenceTo := TRUE;
END_METHOD

PROPERTY PUBLIC Value : ETcVnSvmSgdClassifierType
GET
Value := activeData;
END_GET
SET
activeData := Value;
END_SET
END_PROPERTY

END_FUNCTION_BLOCK

// ---- Datatypes/Enums/_ETcVnTemplateMatchMethod.TcPOU
{attribute 'linkalways'} 
{attribute 'no_explicit_call' := 'This FB is a CLASS and must be accessed using methods or properties'}
{attribute 'enable_dynamic_creation'}
FUNCTION_BLOCK _ETcVnTemplateMatchMethod EXTENDS EnumDatatypeBase
VAR
	localData : ETcVnTemplateMatchMethod;
	activeData : REFERENCE TO ETcVnTemplateMatchMethod;
	enumBaseDatatype : _DINT(localData);
END_VAR

METHOD PRIVATE AddLocalEnumeration
VAR_INPUT
	Enumeration : T_MAXSTRING;
	Value : ETcVnTemplateMatchMethod;
END_VAR
AddEnumeration(Enumeration, Value);
END_METHOD

PROPERTY PUBLIC Address : PVOID
GET
Address := ADR(activeData);
END_GET
END_PROPERTY

METHOD PUBLIC ClearReference
VAR_INPUT
END_VAR
activeData REF= localData;
SetBaseDatatypeReference();
END_METHOD

METHOD PUBLIC Clone : I_Datatype
VAR
    pClone : POINTER TO _ETcVnTemplateMatchMethod;
END_VAR
pClone := __NEW(_ETcVnTemplateMatchMethod(InitialValue := Value));
Clone := pClone^;
END_METHOD

METHOD FB_init : BOOL
VAR_INPUT
	bInitRetains : BOOL; // if TRUE, the retain variables are initialized (warm start / cold start)
	bInCopyCode : BOOL;  // if TRUE, the instance afterwards gets moved into the copy code (online change)
	InitialValue : ETcVnTemplateMatchMethod;
END_VAR
localData := InitialValue;
AddBaseDatatype(enumBaseDatatype);
ClearReference();

AddLocalEnumeration('TCVN_TMM_SQDIFF', ETcVnTemplateMatchMethod.TCVN_TMM_SQDIFF);
AddLocalEnumeration('TCVN_TMM_SQDIFF_NORMED', ETcVnTemplateMatchMethod.TCVN_TMM_SQDIFF_NORMED);
AddLocalEnumeration('TCVN_TMM_CCORR', ETcVnTemplateMatchMethod.TCVN_TMM_CCORR);
AddLocalEnumeration('TCVN_TMM_CCORR_NORMED', ETcVnTemplateMatchMethod.TCVN_TMM_CCORR_NORMED);
AddLocalEnumeration('TCVN_TMM_CCOEFF', ETcVnTemplateMatchMethod.TCVN_TMM_CCOEFF);
AddLocalEnumeration('TCVN_TMM_CCOEFF_NORMED', ETcVnTemplateMatchMethod.TCVN_TMM_CCOEFF_NORMED);
END_METHOD

PROPERTY PUBLIC Identifier : T_MAXSTRING
GET
Identifier := 'ETcVnTemplateMatchMethod';
END_GET
END_PROPERTY

METHOD IsEnumeratorValueEqual : BOOL
VAR_INPUT
	Enumerator : I_KeyValueForwardEnumerator;
END_VAR
VAR
	storedValue : ETcVnTemplateMatchMethod;
END_VAR
IF NOT Enumerator.TryGet(storedValue) THEN
	RETURN;
END_IF

IsEnumeratorValueEqual := storedValue = activeData;
END_METHOD

METHOD PUBLIC MakeReferenceTo
VAR_INPUT
	ReferenceTarget : REFERENCE TO ETcVnTemplateMatchMethod;
END_VAR
activeData REF= ReferenceTarget;
SetBaseDatatypeReference();
END_METHOD

METHOD PROTECTED SetBaseDatatypeReference
VAR_INPUT
END_VAR
enumBaseDatatype.MakeReferenceTo(activeData);
END_METHOD

PROPERTY PUBLIC Size : UDINT
GET
Size := SIZEOF(activeData);
END_GET
END_PROPERTY

METHOD TryMakeReferenceTo : BOOL
VAR_INPUT
	Target : I_Datatype;
END_VAR
VAR
	pTargetData : POINTER TO ETcVnTemplateMatchMethod;
END_VAR
IF NOT IsEquivalentTo(Target) THEN
	RETURN;
END_IF

pTargetData := Target.Address;
activeData REF= pTargetData^;
SetBaseDatatypeReference();
TryMakeReferenceTo := TRUE;
END_METHOD

PROPERTY PUBLIC Value : ETcVnTemplateMatchMethod
GET
Value := activeData;
END_GET
SET
activeData := Value;
END_SET
END_PROPERTY

END_FUNCTION_BLOCK

// ---- Datatypes/Enums/_ETcVnThresholdType.TcPOU
{attribute 'linkalways'} 
{attribute 'no_explicit_call' := 'This FB is a CLASS and must be accessed using methods or properties'}
{attribute 'enable_dynamic_creation'}
FUNCTION_BLOCK _ETcVnThresholdType EXTENDS EnumDatatypeBase
VAR
	localData : ETcVnThresholdType;
	activeData : REFERENCE TO ETcVnThresholdType;
	enumBaseDatatype : _DINT(localData);
END_VAR

METHOD PRIVATE AddLocalEnumeration
VAR_INPUT
	Enumeration : T_MAXSTRING;
	Value : ETcVnThresholdType;
END_VAR
AddEnumeration(Enumeration, Value);
END_METHOD

PROPERTY PUBLIC Address : PVOID
GET
Address := ADR(activeData);
END_GET
END_PROPERTY

METHOD PUBLIC ClearReference
VAR_INPUT
END_VAR
activeData REF= localData;
SetBaseDatatypeReference();
END_METHOD

METHOD PUBLIC Clone : I_Datatype
VAR
    pClone : POINTER TO _ETcVnThresholdType;
END_VAR
pClone := __NEW(_ETcVnThresholdType(InitialValue := Value));
Clone := pClone^;
END_METHOD

METHOD FB_init : BOOL
VAR_INPUT
	bInitRetains : BOOL; // if TRUE, the retain variables are initialized (warm start / cold start)
	bInCopyCode : BOOL;  // if TRUE, the instance afterwards gets moved into the copy code (online change)
	InitialValue : ETcVnThresholdType;
END_VAR
localData := InitialValue;
AddBaseDatatype(enumBaseDatatype);
ClearReference();

AddLocalEnumeration('TCVN_TT_BINARY', ETcVnThresholdType.TCVN_TT_BINARY);
AddLocalEnumeration('TCVN_TT_BINARY_INV', ETcVnThresholdType.TCVN_TT_BINARY_INV);
AddLocalEnumeration('TCVN_TT_TRUNC', ETcVnThresholdType.TCVN_TT_TRUNC);
AddLocalEnumeration('TCVN_TT_TOZERO', ETcVnThresholdType.TCVN_TT_TOZERO);
AddLocalEnumeration('TCVN_TT_TOZERO_INV', ETcVnThresholdType.TCVN_TT_TOZERO_INV);
AddLocalEnumeration('TCVN_TT_OTSU_BINARY', ETcVnThresholdType.TCVN_TT_OTSU_BINARY);
AddLocalEnumeration('TCVN_TT_OTSU_BINARY_INV', ETcVnThresholdType.TCVN_TT_OTSU_BINARY_INV);
AddLocalEnumeration('TCVN_TT_OTSU_TRUNC', ETcVnThresholdType.TCVN_TT_OTSU_TRUNC);
AddLocalEnumeration('TCVN_TT_OTSU_TOZERO', ETcVnThresholdType.TCVN_TT_OTSU_TOZERO);
AddLocalEnumeration('TCVN_TT_OTSU_TOZERO_INV', ETcVnThresholdType.TCVN_TT_OTSU_TOZERO_INV);
AddLocalEnumeration('TCVN_TT_TRIANGLE_BINARY', ETcVnThresholdType.TCVN_TT_TRIANGLE_BINARY);
AddLocalEnumeration('TCVN_TT_TRIANGLE_BINARY_INV', ETcVnThresholdType.TCVN_TT_TRIANGLE_BINARY_INV);
AddLocalEnumeration('TCVN_TT_TRIANGLE_TRUNC', ETcVnThresholdType.TCVN_TT_TRIANGLE_TRUNC);
AddLocalEnumeration('TCVN_TT_TRIANGLE_TOZERO', ETcVnThresholdType.TCVN_TT_TRIANGLE_TOZERO);
AddLocalEnumeration('TCVN_TT_TRIANGLE_TOZERO_INV', ETcVnThresholdType.TCVN_TT_TRIANGLE_TOZERO_INV);
END_METHOD

PROPERTY PUBLIC Identifier : T_MAXSTRING
GET
Identifier := 'ETcVnThresholdType';
END_GET
END_PROPERTY

METHOD IsEnumeratorValueEqual : BOOL
VAR_INPUT
	Enumerator : I_KeyValueForwardEnumerator;
END_VAR
VAR
	storedValue : ETcVnThresholdType;
END_VAR
IF NOT Enumerator.TryGet(storedValue) THEN
	RETURN;
END_IF

IsEnumeratorValueEqual := storedValue = activeData;
END_METHOD

METHOD PUBLIC MakeReferenceTo
VAR_INPUT
	ReferenceTarget : REFERENCE TO ETcVnThresholdType;
END_VAR
activeData REF= ReferenceTarget;
SetBaseDatatypeReference();
END_METHOD

METHOD PROTECTED SetBaseDatatypeReference
VAR_INPUT
END_VAR
enumBaseDatatype.MakeReferenceTo(activeData);
END_METHOD

PROPERTY PUBLIC Size : UDINT
GET
Size := SIZEOF(activeData);
END_GET
END_PROPERTY

METHOD TryMakeReferenceTo : BOOL
VAR_INPUT
	Target : I_Datatype;
END_VAR
VAR
	targetAsEnum : I_EnumDatatype;
	pTargetData : POINTER TO ETcVnThresholdType;
END_VAR
IF NOT Target.TryResolveAsEnumDatatype(targetAsEnum) THEN
	RETURN;
END_IF

IF targetAsEnum.Identifier <> Identifier THEN
	RETURN;
END_IF

pTargetData := Target.Address;
activeData REF= pTargetData^;
SetBaseDatatypeReference();
TryMakeReferenceTo := TRUE;
END_METHOD

PROPERTY PUBLIC Value : ETcVnThresholdType
GET
Value := activeData;
END_GET
SET
activeData := Value;
END_SET
END_PROPERTY

END_FUNCTION_BLOCK

// ---- Datatypes/Enums/_ETcVnVectorCompareMethod.TcPOU
{attribute 'linkalways'} 
{attribute 'no_explicit_call' := 'This FB is a CLASS and must be accessed using methods or properties'}
{attribute 'enable_dynamic_creation'}
FUNCTION_BLOCK _ETcVnVectorCompareMethod EXTENDS EnumDatatypeBase
VAR
	localData : ETcVnVectorCompareMethod;
	activeData : REFERENCE TO ETcVnVectorCompareMethod;
	enumBaseDatatype : _DINT(localData);
END_VAR

METHOD PRIVATE AddLocalEnumeration
VAR_INPUT
	Enumeration : T_MAXSTRING;
	Value : ETcVnVectorCompareMethod;
END_VAR
AddEnumeration(Enumeration, Value);
END_METHOD

PROPERTY PUBLIC Address : PVOID
GET
Address := ADR(activeData);
END_GET
END_PROPERTY

METHOD PUBLIC ClearReference
VAR_INPUT
END_VAR
activeData REF= localData;
SetBaseDatatypeReference();
END_METHOD

METHOD PUBLIC Clone : I_Datatype
VAR
    pClone : POINTER TO _ETcVnVectorCompareMethod;
END_VAR
pClone := __NEW(_ETcVnVectorCompareMethod(InitialValue := Value));
Clone := pClone^;
END_METHOD

METHOD FB_init : BOOL
VAR_INPUT
	bInitRetains : BOOL; // if TRUE, the retain variables are initialized (warm start / cold start)
	bInCopyCode : BOOL;  // if TRUE, the instance afterwards gets moved into the copy code (online change)
	InitialValue : ETcVnVectorCompareMethod;
END_VAR
localData := InitialValue;
AddBaseDatatype(enumBaseDatatype);
ClearReference();

AddLocalEnumeration('TCVN_VCM_EUCLIDEAN', ETcVnVectorCompareMethod.TCVN_VCM_EUCLIDEAN);
AddLocalEnumeration('TCVN_VCM_ELEMENTWISE', ETcVnVectorCompareMethod.TCVN_VCM_ELEMENTWISE);
END_METHOD

PROPERTY PUBLIC Identifier : T_MAXSTRING
GET
Identifier := 'ETcVnVectorCompareMethod';
END_GET
END_PROPERTY

METHOD IsEnumeratorValueEqual : BOOL
VAR_INPUT
	Enumerator : I_KeyValueForwardEnumerator;
END_VAR
VAR
	storedValue : ETcVnVectorCompareMethod;
END_VAR
IF NOT Enumerator.TryGet(storedValue) THEN
	RETURN;
END_IF

IsEnumeratorValueEqual := storedValue = activeData;
END_METHOD

METHOD PUBLIC MakeReferenceTo
VAR_INPUT
	ReferenceTarget : REFERENCE TO ETcVnVectorCompareMethod;
END_VAR
activeData REF= ReferenceTarget;
SetBaseDatatypeReference();
END_METHOD

METHOD PROTECTED SetBaseDatatypeReference
VAR_INPUT
END_VAR
enumBaseDatatype.MakeReferenceTo(activeData);
END_METHOD

PROPERTY PUBLIC Size : UDINT
GET
Size := SIZEOF(activeData);
END_GET
END_PROPERTY

METHOD TryMakeReferenceTo : BOOL
VAR_INPUT
	Target : I_Datatype;
END_VAR
VAR
	pTargetData : POINTER TO ETcVnVectorCompareMethod;
END_VAR
IF NOT IsEquivalentTo(Target) THEN
	RETURN;
END_IF

pTargetData := Target.Address;
activeData REF= pTargetData^;
SetBaseDatatypeReference();
TryMakeReferenceTo := TRUE;
END_METHOD

PROPERTY PUBLIC Value : ETcVnVectorCompareMethod
GET
Value := activeData;
END_GET
SET
activeData := Value;
END_SET
END_PROPERTY

END_FUNCTION_BLOCK

// ---- Datatypes/Enums/_ETcVnWorldCoordinateSystem.TcPOU
{attribute 'linkalways'} 
{attribute 'no_explicit_call' := 'This FB is a CLASS and must be accessed using methods or properties'}
{attribute 'enable_dynamic_creation'}
FUNCTION_BLOCK _ETcVnWorldCoordinateSystem EXTENDS EnumDatatypeBase
VAR
	localData : ETcVnWorldCoordinateSystem;
	activeData : REFERENCE TO ETcVnWorldCoordinateSystem;
	enumBaseDatatype : _DINT(localData);
END_VAR

METHOD PRIVATE AddLocalEnumeration
VAR_INPUT
	Enumeration : T_MAXSTRING;
	Value : ETcVnWorldCoordinateSystem;
END_VAR
AddEnumeration(Enumeration, Value);
END_METHOD

PROPERTY PUBLIC Address : PVOID
GET
Address := ADR(activeData);
END_GET
END_PROPERTY

METHOD PUBLIC ClearReference
VAR_INPUT
END_VAR
activeData REF= localData;
SetBaseDatatypeReference();
END_METHOD

METHOD PUBLIC Clone : I_Datatype
VAR
    pClone : POINTER TO _ETcVnWorldCoordinateSystem;
END_VAR
pClone := __NEW(_ETcVnWorldCoordinateSystem(InitialValue := Value));
Clone := pClone^;
END_METHOD

METHOD FB_init : BOOL
VAR_INPUT
	bInitRetains : BOOL; // if TRUE, the retain variables are initialized (warm start / cold start)
	bInCopyCode : BOOL;  // if TRUE, the instance afterwards gets moved into the copy code (online change)
	InitialValue : ETcVnWorldCoordinateSystem;
END_VAR
localData := InitialValue;
AddBaseDatatype(enumBaseDatatype);
ClearReference();

AddLocalEnumeration('TCVN_WCS_X_RIGHT_Y_DOWN' , ETcVnWorldCoordinateSystem.TCVN_WCS_X_RIGHT_Y_DOWN);
AddLocalEnumeration('TCVN_WCS_X_DOWN_Y_RIGHT', ETcVnWorldCoordinateSystem.TCVN_WCS_X_DOWN_Y_RIGHT);
AddLocalEnumeration('TCVN_WCS_X_LEFT_Y_DOWN', ETcVnWorldCoordinateSystem.TCVN_WCS_X_LEFT_Y_DOWN);
AddLocalEnumeration('TCVN_WCS_X_UP_Y_RIGHT', ETcVnWorldCoordinateSystem.TCVN_WCS_X_UP_Y_RIGHT);
AddLocalEnumeration('TCVN_WCS_X_RIGHT_Y_UP', ETcVnWorldCoordinateSystem.TCVN_WCS_X_RIGHT_Y_UP);
AddLocalEnumeration('TCVN_WCS_X_DOWN_Y_LEFT', ETcVnWorldCoordinateSystem.TCVN_WCS_X_DOWN_Y_LEFT);
AddLocalEnumeration('TCVN_WCS_X_LEFT_Y_UP', ETcVnWorldCoordinateSystem.TCVN_WCS_X_LEFT_Y_UP);
AddLocalEnumeration('TCVN_WCS_X_UP_Y_LEFT', ETcVnWorldCoordinateSystem.TCVN_WCS_X_UP_Y_LEFT);
END_METHOD

PROPERTY PUBLIC Identifier : T_MAXSTRING
GET
Identifier := 'ETcVnWorldCoordinateSystem';
END_GET
END_PROPERTY

METHOD IsEnumeratorValueEqual : BOOL
VAR_INPUT
	Enumerator : I_KeyValueForwardEnumerator;
END_VAR
VAR
	storedValue : ETcVnWorldCoordinateSystem;
END_VAR
IF NOT Enumerator.TryGet(storedValue) THEN
	RETURN;
END_IF

IsEnumeratorValueEqual := storedValue = activeData;
END_METHOD

METHOD PUBLIC MakeReferenceTo
VAR_INPUT
	ReferenceTarget : REFERENCE TO ETcVnWorldCoordinateSystem;
END_VAR
activeData REF= ReferenceTarget;
SetBaseDatatypeReference();
END_METHOD

METHOD PROTECTED SetBaseDatatypeReference
VAR_INPUT
END_VAR
enumBaseDatatype.MakeReferenceTo(activeData);
END_METHOD

PROPERTY PUBLIC Size : UDINT
GET
Size := SIZEOF(activeData);
END_GET
END_PROPERTY

METHOD TryMakeReferenceTo : BOOL
VAR_INPUT
	Target : I_Datatype;
END_VAR
VAR
	pTargetData : POINTER TO ETcVnWorldCoordinateSystem;
END_VAR
IF NOT IsEquivalentTo(Target) THEN
	RETURN;
END_IF

pTargetData := Target.Address;
activeData REF= pTargetData^;
SetBaseDatatypeReference();
TryMakeReferenceTo := TRUE;
END_METHOD

PROPERTY PUBLIC Value : ETcVnWorldCoordinateSystem
GET
Value := activeData;
END_GET
SET
activeData := Value;
END_SET
END_PROPERTY

END_FUNCTION_BLOCK

// ---- Datatypes/Enums/_ETcWatchdogAccumulationType.TcPOU
{attribute 'linkalways'} 
{attribute 'no_explicit_call' := 'This FB is a CLASS and must be accessed using methods or properties'}
{attribute 'enable_dynamic_creation'}
FUNCTION_BLOCK _ETcWatchdogAccumulationType EXTENDS EnumDatatypeBase
VAR
	localData : ETcWatchdogAccumulationType;
	activeData : REFERENCE TO ETcWatchdogAccumulationType;
	enumBaseDatatype : _UINT(localData);
END_VAR

METHOD PRIVATE AddLocalEnumeration
VAR_INPUT
	Enumeration : T_MAXSTRING;
	Value : ETcWatchdogAccumulationType;
END_VAR
AddEnumeration(Enumeration, Value);
END_METHOD

PROPERTY PUBLIC Address : PVOID
GET
Address := ADR(activeData);
END_GET
END_PROPERTY

METHOD PUBLIC ClearReference
VAR_INPUT
END_VAR
activeData REF= localData;
SetBaseDatatypeReference();
END_METHOD

METHOD PUBLIC Clone : I_Datatype
VAR
    pClone : POINTER TO _ETcWatchdogAccumulationType;
END_VAR
pClone := __NEW(_ETcWatchdogAccumulationType(InitialValue := Value));
Clone := pClone^;
END_METHOD

METHOD FB_init : BOOL
VAR_INPUT
	bInitRetains : BOOL; // if TRUE, the retain variables are initialized (warm start / cold start)
	bInCopyCode : BOOL;  // if TRUE, the instance afterwards gets moved into the copy code (online change)
	InitialValue : ETcWatchdogAccumulationType;
END_VAR
localData := InitialValue;
AddBaseDatatype(enumBaseDatatype);
ClearReference();

AddLocalEnumeration('WD_ACC_TYPE_MEAN', ETcWatchdogAccumulationType.WD_ACC_TYPE_MEAN);
AddLocalEnumeration('WD_ACC_TYPE_PRODUCT', ETcWatchdogAccumulationType.WD_ACC_TYPE_PRODUCT);
END_METHOD

PROPERTY PUBLIC Identifier : T_MAXSTRING
GET
Identifier := 'ETcWatchdogAccumulationType';
END_GET
END_PROPERTY

METHOD IsEnumeratorValueEqual : BOOL
VAR_INPUT
	Enumerator : I_KeyValueForwardEnumerator;
END_VAR
VAR
	storedValue : ETcWatchdogAccumulationType;
END_VAR
IF NOT Enumerator.TryGet(storedValue) THEN
	RETURN;
END_IF

IsEnumeratorValueEqual := storedValue = activeData;
END_METHOD

METHOD PUBLIC MakeReferenceTo
VAR_INPUT
	ReferenceTarget : REFERENCE TO ETcWatchdogAccumulationType;
END_VAR
activeData REF= ReferenceTarget;
SetBaseDatatypeReference();
END_METHOD

METHOD PROTECTED SetBaseDatatypeReference
VAR_INPUT
END_VAR
enumBaseDatatype.MakeReferenceTo(activeData);
END_METHOD

PROPERTY PUBLIC Size : UDINT
GET
Size := SIZEOF(activeData);
END_GET
END_PROPERTY

METHOD TryMakeReferenceTo : BOOL
VAR_INPUT
	Target : I_Datatype;
END_VAR
VAR
	pTargetData : POINTER TO ETcWatchdogAccumulationType;
END_VAR
IF NOT IsEquivalentTo(Target) THEN
	RETURN;
END_IF

pTargetData := Target.Address;
activeData REF= pTargetData^;
SetBaseDatatypeReference();
TryMakeReferenceTo := TRUE;
END_METHOD

PROPERTY PUBLIC Value : ETcWatchdogAccumulationType
GET
Value := activeData;
END_GET
SET
activeData := Value;
END_SET
END_PROPERTY

END_FUNCTION_BLOCK

// ---- Datatypes/Enums/_GEV_CAMERA_STATE.TcPOU
{attribute 'linkalways'} 
{attribute 'no_explicit_call' := 'This FB is a CLASS and must be accessed using methods or properties'}
{attribute 'enable_dynamic_creation'}
FUNCTION_BLOCK _GEV_CAMERA_STATE EXTENDS EnumDatatypeBase
VAR
	localData : GEV_CAMERA_STATE;
	activeData : REFERENCE TO GEV_CAMERA_STATE;
	enumBaseDatatype : _BYTE(localData);
END_VAR

METHOD PRIVATE AddLocalEnumeration
VAR_INPUT
	Enumeration : T_MAXSTRING;
	Value : GEV_CAMERA_STATE;
END_VAR
AddEnumeration(Enumeration, Value);
END_METHOD

PROPERTY PUBLIC Address : PVOID
GET
Address := ADR(activeData);
END_GET
END_PROPERTY

METHOD PUBLIC ClearReference
VAR_INPUT
END_VAR
activeData REF= localData;
SetBaseDatatypeReference();
END_METHOD

METHOD PUBLIC Clone : I_Datatype
VAR
    pClone : POINTER TO _GEV_CAMERA_STATE;
END_VAR
pClone := __NEW(_GEV_CAMERA_STATE(InitialValue := Value));
Clone := pClone^;
END_METHOD

METHOD FB_init : BOOL
VAR_INPUT
	bInitRetains : BOOL; // if TRUE, the retain variables are initialized (warm start / cold start)
	bInCopyCode : BOOL;  // if TRUE, the instance afterwards gets moved into the copy code (online change)
	InitialValue : GEV_CAMERA_STATE;
END_VAR
localData := InitialValue;
AddBaseDatatype(enumBaseDatatype);
ClearReference();

AddLocalEnumeration('GEV_CAMERA_IDLE', GEV_CAMERA_STATE.GEV_CAMERA_IDLE);
AddLocalEnumeration('GEV_CONTROL_CHANNEL_OPEN_MASK', GEV_CAMERA_STATE.GEV_CONTROL_CHANNEL_OPEN_MASK);
AddLocalEnumeration('GEV_STREAM_CHANNELS_OPEN_MASK', GEV_CAMERA_STATE.GEV_STREAM_CHANNELS_OPEN_MASK);
AddLocalEnumeration('GEV_CONTROL_CHANNEL_OPEN', GEV_CAMERA_STATE.GEV_CONTROL_CHANNEL_OPEN);
AddLocalEnumeration('GEV_STREAM_CHANNELS_OPEN', GEV_CAMERA_STATE.GEV_STREAM_CHANNELS_OPEN);
END_METHOD

PROPERTY PUBLIC Identifier : T_MAXSTRING
GET
Identifier := 'GEV_CAMERA_STATE';
END_GET
END_PROPERTY

METHOD IsEnumeratorValueEqual : BOOL
VAR_INPUT
	Enumerator : I_KeyValueForwardEnumerator;
END_VAR
VAR
	storedValue : GEV_CAMERA_STATE;
END_VAR
IF NOT Enumerator.TryGet(storedValue) THEN
	RETURN;
END_IF

IsEnumeratorValueEqual := storedValue = activeData;
END_METHOD

METHOD PUBLIC MakeReferenceTo
VAR_INPUT
	ReferenceTarget : REFERENCE TO GEV_CAMERA_STATE;
END_VAR
activeData REF= ReferenceTarget;
SetBaseDatatypeReference();
END_METHOD

METHOD PROTECTED SetBaseDatatypeReference
VAR_INPUT
END_VAR
enumBaseDatatype.MakeReferenceTo(activeData);
END_METHOD

PROPERTY PUBLIC Size : UDINT
GET
Size := SIZEOF(activeData);
END_GET
END_PROPERTY

METHOD TryMakeReferenceTo : BOOL
VAR_INPUT
	Target : I_Datatype;
END_VAR
VAR
	targetAsEnum : I_EnumDatatype;
	pTargetData : POINTER TO GEV_CAMERA_STATE;
END_VAR
IF NOT Target.TryResolveAsEnumDatatype(targetAsEnum) THEN
	RETURN;
END_IF

IF targetAsEnum.Identifier <> Identifier THEN
	RETURN;
END_IF

pTargetData := Target.Address;
activeData REF= pTargetData^;
SetBaseDatatypeReference();
TryMakeReferenceTo := TRUE;
END_METHOD

PROPERTY PUBLIC Value : GEV_CAMERA_STATE
GET
Value := activeData;
END_GET
SET
activeData := Value;
END_SET
END_PROPERTY

END_FUNCTION_BLOCK

// ---- Datatypes/Interfaces/_ITcVnContainer.TcPOU
{attribute 'linkalways'} 
{attribute 'no_explicit_call' := 'This FB is a CLASS and must be accessed using methods or properties'}
{attribute 'enable_dynamic_creation'}
FUNCTION_BLOCK _ITcVnContainer EXTENDS InterfaceDatatypeBase
VAR
	localData : ITcVnContainer;
	activeData : REFERENCE TO ITcVnContainer REF= localData;
END_VAR

PROPERTY PUBLIC Address : PVOID
GET
Address := ADR(activeData);
END_GET
END_PROPERTY

METHOD PUBLIC ClearReference
VAR_INPUT
END_VAR
activeData REF= localData;
END_METHOD

METHOD PUBLIC Clone : I_Datatype
VAR
    pClone : POINTER TO _ITcVnContainer;
END_VAR
pClone := __NEW(_ITcVnContainer);
Clone := pClone^;
END_METHOD

METHOD FB_exit : BOOL
VAR_INPUT
	bInCopyCode : BOOL; // if TRUE, the exit method is called for exiting an instance that is copied afterwards (online change).
END_VAR
IF bInCopyCode THEN
	RETURN;
END_IF

TryTcReleaseLocal();
END_METHOD

METHOD PUBLIC HasType : BOOL
VAR_INPUT
	ContainerType : GUID;
END_VAR
VAR
    actualGuid : GUID;
END_VAR
IF NOT IsValid THEN
    RETURN;
END_IF

IF NOT SUCCEEDED(activeData.GetTypeGuid(actualGuid)) THEN
    RETURN;
END_IF

IF NOT (GuidsEqualByVal(ContainerType, actualGuid)) THEN
	RETURN;
END_IF

HasType := TRUE;
END_METHOD

PROPERTY PUBLIC Identifier : T_MAXSTRING
GET
Identifier := 'ITcVnContainer';
END_GET
END_PROPERTY

PROPERTY PUBLIC IsValid : BOOL
GET
IsValid := activeData <> 0;
END_GET
END_PROPERTY

METHOD PUBLIC MakeReferenceTo
VAR_INPUT
	ReferenceTarget : REFERENCE TO ITcVnContainer;
END_VAR
activeData REF= ReferenceTarget;
END_METHOD

METHOD PRIVATE Serialize_ContainerType_Vector_DINT
VAR_INPUT
	Serializer : I_Serializer;
END_VAR
VAR
	hr : HRESULT;
	_value : _DINT(0);
	elementCount : ULINT;
	i : ULINT;
END_VAR
activeData.GetElementNum(elementCount);

FOR i := 0 TO elementCount - 1 DO 
	
	hr := F_VN_GetAt_DINT(activeData, _value.Value, i, S_OK);
	
	IF SUCCEEDED(hr) THEN
		Serializer.AddObject(_value);
	ELSE
		Serializer.AddNull();
	END_IF
	
END_FOR
END_METHOD

METHOD PRIVATE Serialize_ContainerType_Vector_INT
VAR_INPUT
	Serializer : I_Serializer;
END_VAR
VAR
	hr : HRESULT;
	_value : _INT(0);
	elementCount : ULINT;
	i : ULINT;
END_VAR
activeData.GetElementNum(elementCount);

FOR i := 0 TO elementCount - 1 DO 
	
	hr := F_VN_GetAt_INT(activeData, _value.Value, i, S_OK);
	
	IF SUCCEEDED(hr) THEN
		Serializer.AddObject(_value);
	ELSE
		Serializer.AddNull();
	END_IF
	
END_FOR
END_METHOD

METHOD PRIVATE Serialize_ContainerType_Vector_ITcVnImage
VAR_INPUT
	Serializer : I_Serializer;
END_VAR
VAR
	hr : HRESULT;
	_value : _ITcVnImage;
	elementCount : ULINT;
	i : ULINT;
END_VAR
activeData.GetElementNum(elementCount);

FOR i := 0 TO elementCount - 1 DO 
	
	hr := F_VN_GetAt_ITcVnImage(activeData, _value.Value, i, S_OK);
	
	IF SUCCEEDED(hr) THEN
		Serializer.AddObject(_value);
	ELSE
		Serializer.AddNull();
	END_IF
	
END_FOR
END_METHOD

METHOD PRIVATE Serialize_ContainerType_Vector_LREAL
VAR_INPUT
	Serializer : I_Serializer;
END_VAR
VAR
	hr : HRESULT;
	_value : _LREAL(0);
	elementCount : ULINT;
	i : ULINT;
END_VAR
activeData.GetElementNum(elementCount);

FOR i := 0 TO elementCount - 1 DO 
	
	hr := F_VN_GetAt_LREAL(activeData, _value.Value, i, S_OK);
	
	IF SUCCEEDED(hr) THEN
		Serializer.AddObject(_value);
	ELSE
		Serializer.AddNull();
	END_IF
	
END_FOR
END_METHOD

METHOD PRIVATE Serialize_ContainerType_Vector_REAL
VAR_INPUT
	Serializer : I_Serializer;
END_VAR
VAR
	hr : HRESULT;
	_value : _REAL(0);
	elementCount : ULINT;
	i : ULINT;
END_VAR
activeData.GetElementNum(elementCount);

FOR i := 0 TO elementCount - 1 DO 
	
	hr := F_VN_GetAt_REAL(activeData, _value.Value, i, S_OK);
	
	IF SUCCEEDED(hr) THEN
		Serializer.AddObject(_value);
	ELSE
		Serializer.AddNull();
	END_IF
	
END_FOR
END_METHOD

METHOD PRIVATE Serialize_ContainerType_Vector_SINT
VAR_INPUT
	Serializer : I_Serializer;
END_VAR
VAR
	hr : HRESULT;
	_value : _SINT(0);
	elementCount : ULINT;
	i : ULINT;
END_VAR
activeData.GetElementNum(elementCount);

FOR i := 0 TO elementCount - 1 DO 
	
	hr := F_VN_GetAt_SINT(activeData, _value.Value, i, S_OK);
	
	IF SUCCEEDED(hr) THEN
		Serializer.AddObject(_value);
	ELSE
		Serializer.AddNull();
	END_IF
	
END_FOR
END_METHOD

METHOD PRIVATE Serialize_ContainerType_Vector_UDINT
VAR_INPUT
	Serializer : I_Serializer;
END_VAR
VAR
	hr : HRESULT;
	_value : _ULINT(0);
	elementCount : ULINT;
	i : ULINT;
END_VAR
activeData.GetElementNum(elementCount);

FOR i := 0 TO elementCount - 1 DO 
	
	hr := F_VN_GetAt_ULINT(activeData, _value.Value, i, S_OK);
	
	IF SUCCEEDED(hr) THEN
		Serializer.AddObject(_value);
	ELSE
		Serializer.AddNull();
	END_IF
	
END_FOR
END_METHOD

METHOD PRIVATE Serialize_ContainerType_Vector_UINT
VAR_INPUT
	Serializer : I_Serializer;
END_VAR
VAR
	hr : HRESULT;
	_value : _UINT(0);
	elementCount : ULINT;
	i : ULINT;
END_VAR
activeData.GetElementNum(elementCount);

FOR i := 0 TO elementCount - 1 DO 
	
	hr := F_VN_GetAt_UINT(activeData, _value.Value, i, S_OK);
	
	IF SUCCEEDED(hr) THEN
		Serializer.AddObject(_value);
	ELSE
		Serializer.AddNull();
	END_IF
	
END_FOR
END_METHOD

METHOD PRIVATE Serialize_ContainerType_Vector_ULINT
VAR_INPUT
	Serializer : I_Serializer;
END_VAR
VAR
	hr : HRESULT;
	_value : _ULINT(0);
	elementCount : ULINT;
	i : ULINT;
END_VAR
activeData.GetElementNum(elementCount);

FOR i := 0 TO elementCount - 1 DO 
	
	hr := F_VN_GetAt_ULINT(activeData, _value.Value, i, S_OK);
	
	IF SUCCEEDED(hr) THEN
		Serializer.AddObject(_value);
	ELSE
		Serializer.AddNull();
	END_IF
	
END_FOR
END_METHOD

METHOD PRIVATE Serialize_ContainerType_Vector_USINT
VAR_INPUT
	Serializer : I_Serializer;
END_VAR
VAR
	hr : HRESULT;
	_value : _USINT(0);
	elementCount : ULINT;
	i : ULINT;
END_VAR
activeData.GetElementNum(elementCount);

FOR i := 0 TO elementCount - 1 DO 
	
	hr := F_VN_GetAt_USINT(activeData, _value.Value, i, S_OK);
	
	IF SUCCEEDED(hr) THEN
		Serializer.AddObject(_value);
	ELSE
		Serializer.AddNull();
	END_IF
	
END_FOR
END_METHOD

METHOD PUBLIC SerializeWith
VAR_INPUT
	Serializer : I_Serializer;
END_VAR
VAR
	containerTypeName : _STRING('');
	containerTypeGuid : _GUID;
	elementTypeGuid : _GUID;
    elementNum : _ULINT(0);
    elementSize : _ULINT(0);
END_VAR
IF NOT (activeData <> 0) THEN
	Serializer.AddNull();
	RETURN;
END_IF

activeData.GetTypeName(containerTypeName.Value,UDINT_TO_UINT(containerTypeName.Size));
activeData.GetTypeGuid(containerTypeGuid.Value);
activeData.GetElementTypeGuid(elementTypeGuid.Value);
activeData.GetElementNum(elementNum.Value);
activeData.GetElementSize(elementSize.Value);

Serializer.StartObject();
Serializer.AddKeyObject('containerTypeName', containerTypeName);
Serializer.AddKeyString('containerTypeGuid', containerTypeGuid.ToString());
Serializer.AddKeyString('elementTypeGuid', elementTypeGuid.ToString());
Serializer.AddKeyObject('elementNum', elementNum);
Serializer.AddKeyObject('elementSize', elementSize);
Serializer.AddKey('elements');
Serializer.StartArray();

IF containerTypeName.Value = 'CTcVnContainer_Vector_SINT' THEN
	Serialize_ContainerType_Vector_SINT(Serializer);		
ELSIF containerTypeName.Value = 'CTcVnContainer_Vector_USINT' THEN
	Serialize_ContainerType_Vector_USINT(Serializer);
ELSIF containerTypeName.Value = 'CTcVnContainer_Vector_INT' THEN
	Serialize_ContainerType_Vector_INT(Serializer);
ELSIF containerTypeName.Value = 'CTcVnContainer_Vector_UINT' THEN
	Serialize_ContainerType_Vector_UINT(Serializer);
ELSIF containerTypeName.Value = 'CTcVnContainer_Vector_DINT' THEN
	Serialize_ContainerType_Vector_DINT(Serializer);
ELSIF containerTypeName.Value = 'CTcVnContainer_Vector_UDINT' THEN
	Serialize_ContainerType_Vector_UDINT(Serializer);
ELSIF containerTypeName.Value = 'CTcVnContainer_Vector_ULINT' THEN
	Serialize_ContainerType_Vector_ULINT(Serializer);
ELSIF containerTypeName.Value = 'CTcVnContainer_Vector_REAL' THEN
	Serialize_ContainerType_Vector_REAL(Serializer);
ELSIF containerTypeName.Value = 'CTcVnContainer_Vector_LREAL' THEN
	Serialize_ContainerType_Vector_LREAL(Serializer);
ELSIF containerTypeName.Value = 'CTcVnContainer_Vector_ITcVnImage' THEN
	Serialize_ContainerType_Vector_ITcVnImage(Serializer);
//ELSIF containerTypeName.Value = 'CTcVnContainer_Vector_' THEN
//	Serialize_ContainerType_Vector_(Serializer);
//ELSIF containerTypeName.Value = 'CTcVnContainer_Vector_' THEN
//	Serialize_ContainerType_Vector_(Serializer);
//ELSIF containerTypeName.Value = 'CTcVnContainer_Vector_' THEN
//	Serialize_ContainerType_Vector_(Serializer);
//ELSIF containerTypeName.Value = 'CTcVnContainer_Vector_' THEN
//	Serialize_ContainerType_Vector_(Serializer);
//ELSIF containerTypeName.Value = 'CTcVnContainer_Vector_' THEN
//	Serialize_ContainerType_Vector_(Serializer);
//ELSIF containerTypeName.Value = 'CTcVnContainer_Vector_' THEN
//	Serialize_ContainerType_Vector_(Serializer);	
		
END_IF
Serializer.EndArray();
Serializer.EndObject();
END_METHOD

PROPERTY PUBLIC Size : UDINT
GET
Size := SIZEOF(activeData);
END_GET
END_PROPERTY

METHOD TryDeserializeFrom : BOOL
VAR_INPUT
	Deserializer : I_Deserializer;
	Feedback : I_DeserializerFeedback;
END_VAR
VAR
END_VAR
// not yet implemented.  This will just be a reverse of the serialization code.
END_METHOD

METHOD PUBLIC TryGetTypeName : BOOL
VAR_INPUT
	Destination : REFERENCE TO STRING;
END_VAR
IF NOT IsValid THEN
	RETURN;
END_IF

TryGetTypeName := SUCCEEDED(activeData.GetTypeName(Destination, 255));
END_METHOD

METHOD TryMakeReferenceTo : BOOL
VAR_INPUT
	Target : I_Datatype;
END_VAR
VAR
	pTargetData : POINTER TO ITcVnContainer;
END_VAR
IF NOT IsEquivalentTo(Target) THEN
	RETURN;
END_IF

pTargetData := Target.Address;
activeData REF= pTargetData^;
TryMakeReferenceTo := TRUE;
END_METHOD

METHOD PUBLIC TryTcAddRef : BOOL
VAR_INPUT
END_VAR
IF activeData = 0 THEN
	RETURN;
END_IF

IF activeData.TcAddRef() = 0 THEN
	activeData := 0;
END_IF

TryTcAddRef := TRUE;
END_METHOD

METHOD PUBLIC TryTcRelease : BOOL
VAR_INPUT
END_VAR
IF activeData = 0 THEN
	RETURN;
END_IF

IF activeData.TcRelease() = 0 THEN
	activeData := 0;
END_IF

TryTcRelease := TRUE;
END_METHOD

METHOD PUBLIC TryTcReleaseLocal : BOOL
VAR_INPUT
END_VAR
IF localData = 0 THEN
	RETURN;
END_IF

IF localData.TcRelease() = 0 THEN
	localData := 0;
END_IF

TryTcReleaseLocal := TRUE;
END_METHOD

PROPERTY PUBLIC Value : REFERENCE TO ITcVnContainer
GET
Value REF= activeData;
END_GET
END_PROPERTY

END_FUNCTION_BLOCK

// ---- Datatypes/Structs/_TcVnKeyPoint.TcPOU
{attribute 'linkalways'} 
{attribute 'no_explicit_call' := 'This FB is a CLASS and must be accessed using methods or properties'}
{attribute 'enable_dynamic_creation'}
FUNCTION_BLOCK _TcVnKeyPoint EXTENDS StructuredDatatypeBase
VAR
	localData : TcVnKeyPoint;
	activeData : REFERENCE TO TcVnKeyPoint REF= localData;
    _aPoint : _TcVnPoint2_REAL();
    _fDiameter : _REAL(localdata.fDiameter);
    _fAngle : _REAL(localdata.fAngle);
    _fResponse : _REAL(localdata.fResponse);
    _nOctave : _DINT(localdata.nOctave);
    _nClassId : _DINT(localdata.nClassId);
END_VAR

PROPERTY PUBLIC Address : PVOID
GET
Address := ADR(activeData);
END_GET
END_PROPERTY

PROPERTY PUBLIC aPoint : REFERENCE TO _TcVnPoint2_REAL
GET
aPoint REF= _aPoint;
END_GET
END_PROPERTY

METHOD PUBLIC ClearReference
VAR_INPUT
END_VAR
activeData REF= localData;
SetMemberReference();
END_METHOD

METHOD PUBLIC Clone : I_Datatype
VAR
    pClone : POINTER TO _TcVnKeyPoint;
END_VAR
pClone := __NEW(_TcVnKeyPoint());
pClone^.Value := Value;
Clone := pClone^;
END_METHOD

PROPERTY PUBLIC fAngle : REFERENCE TO _REAL
GET
fAngle REF= _fAngle;
END_GET
END_PROPERTY

METHOD FB_init : BOOL
VAR_INPUT
	bInitRetains : BOOL; // if TRUE, the retain variables are initialized (warm start / cold start)
	bInCopyCode : BOOL;  // if TRUE, the instance afterwards gets moved into the copy code (online change)
END_VAR
SetMemberReference();
AddMember('aPoint', _aPoint);
AddMember('fDiameter', _fDiameter);
AddMember('fAngle', _fAngle);
AddMember('fResponse', _fResponse);
AddMember('nOctave', _nOctave);
AddMember('nClassId', _nClassId);
END_METHOD

PROPERTY PUBLIC fDiameter : REFERENCE TO _REAL
GET
fDiameter REF= _fDiameter;
END_GET
END_PROPERTY

PROPERTY PUBLIC fResponse : REFERENCE TO _REAL
GET
fResponse REF= _fResponse;
END_GET
END_PROPERTY

PROPERTY PUBLIC Identifier : T_MAXSTRING
GET
Identifier := 'TcVnKeyPoint';
END_GET
END_PROPERTY

METHOD PUBLIC MakeReferenceTo
VAR_INPUT
	ReferenceTarget : REFERENCE TO TcVnKeyPoint;
END_VAR
activeData REF= ReferenceTarget;
SetMemberReference();
END_METHOD

PROPERTY PUBLIC nClassId : REFERENCE TO _DINT
GET
nClassId REF= _nClassId;
END_GET
END_PROPERTY

PROPERTY PUBLIC nOctave : REFERENCE TO _DINT
GET
nOctave REF= _nOctave;
END_GET
END_PROPERTY

METHOD PROTECTED SetMemberReference
VAR_INPUT
END_VAR
_aPoint.MakeReferenceTo(activeData.aPoint);
_fDiameter.MakeReferenceTo(activeData.fDiameter);
_fAngle.MakeReferenceTo(activeData.fAngle);
_fResponse.MakeReferenceTo(activeData.fResponse);
_nOctave.MakeReferenceTo(activeData.nOctave);
_nClassId.MakeReferenceTo(activeData.nClassId);
END_METHOD

PROPERTY PUBLIC Size : UDINT
GET
Size := SIZEOF(activeData);
END_GET
END_PROPERTY

METHOD TryMakeReferenceTo : BOOL
VAR_INPUT
	Target : I_Datatype;
END_VAR
VAR
	pTargetData : POINTER TO TcVnKeyPoint;
END_VAR
IF NOT IsEquivalentTo(Target) THEN
	RETURN;
END_IF

pTargetData := Target.Address;
activeData REF= pTargetData^;
SetMemberReference();
TryMakeReferenceTo := TRUE;
END_METHOD

PROPERTY PUBLIC Value : REFERENCE TO TcVnKeyPoint
GET
Value REF= activeData;
END_GET
END_PROPERTY

END_FUNCTION_BLOCK

// ---- Datatypes/Structs/_TcVnParamsKAZE.TcPOU
{attribute 'linkalways'} 
{attribute 'no_explicit_call' := 'This FB is a CLASS and must be accessed using methods or properties'}
{attribute 'enable_dynamic_creation'}
FUNCTION_BLOCK _TcVnParamsKAZE EXTENDS StructuredDatatypeBase
VAR
	localData : TcVnParamsKAZE;
	activeData : REFERENCE TO TcVnParamsKAZE REF= localData;
    _bExtended     : _BOOL(localdata.bExtended);
    _bUpright      : _BOOL(localdata.bUpright);
    _fThreshold    : _REAL(localdata.fThreshold);
    _nOctaves      : _UDINT(localdata.nOctaves);
    _nOctaveLayers : _UDINT(localdata.nOctaveLayers);
    _eDiffusivity  : _ETcVnDiffusivityTypeKAZE(localdata.eDiffusivity);
END_VAR

PROPERTY PUBLIC Address : PVOID
GET
Address := ADR(activeData);
END_GET
END_PROPERTY

PROPERTY PUBLIC bExtended : REFERENCE TO _BOOL
GET
bExtended REF= _bExtended;
END_GET
END_PROPERTY

PROPERTY PUBLIC bUpright : REFERENCE TO _BOOL
GET
bUpright REF= _bUpright;
END_GET
END_PROPERTY

METHOD PUBLIC ClearReference
VAR_INPUT
END_VAR
activeData REF= localData;
SetMemberReference();
END_METHOD

METHOD PUBLIC Clone : I_Datatype
VAR
    pClone : POINTER TO _TcVnParamsKAZE;
END_VAR
pClone := __NEW(_TcVnParamsKAZE());
pClone^.Value := Value;
Clone := pClone^;
END_METHOD

PROPERTY PUBLIC eDiffusivity : REFERENCE TO _ETcVnDiffusivityTypeKAZE
GET
eDiffusivity REF= _eDiffusivity;
END_GET
END_PROPERTY

METHOD FB_init : BOOL
VAR_INPUT
	bInitRetains : BOOL; // if TRUE, the retain variables are initialized (warm start / cold start)
	bInCopyCode : BOOL;  // if TRUE, the instance afterwards gets moved into the copy code (online change)
END_VAR
SetMemberReference();
AddMember('bExtended', _bExtended);
AddMember('bUpright', _bUpright);
AddMember('fThreshold', _fThreshold);
AddMember('nOctaves', _nOctaves);
AddMember('nOctaveLayers', _nOctaveLayers);
AddMember('eDiffusivity', _eDiffusivity);
END_METHOD

PROPERTY PUBLIC fThreshold : REFERENCE TO _REAL
GET
fThreshold REF= _fThreshold;
END_GET
END_PROPERTY

PROPERTY PUBLIC Identifier : T_MAXSTRING
GET
Identifier := 'TcVnParamsKAZE';
END_GET
END_PROPERTY

METHOD PUBLIC MakeReferenceTo
VAR_INPUT
	ReferenceTarget : REFERENCE TO TcVnParamsKAZE;
END_VAR
activeData REF= ReferenceTarget;
SetMemberReference();
END_METHOD

PROPERTY PUBLIC nOctaveLayers : REFERENCE TO _UDINT
GET
nOctaveLayers REF= _nOctaveLayers;
END_GET
END_PROPERTY

PROPERTY PUBLIC nOctaves : REFERENCE TO _UDINT
GET
nOctaves REF= _nOctaves;
END_GET
END_PROPERTY

METHOD PROTECTED SetMemberReference
VAR_INPUT
END_VAR
_bExtended.MakeReferenceTo(activeData.bExtended);
_bUpright.MakeReferenceTo(activeData.bUpright);
_fThreshold.MakeReferenceTo(activeData.fThreshold);
_nOctaves.MakeReferenceTo(activeData.nOctaves);
_nOctaveLayers.MakeReferenceTo(activeData.nOctaveLayers);
_eDiffusivity.MakeReferenceTo(activeData.eDiffusivity);
END_METHOD

PROPERTY PUBLIC Size : UDINT
GET
Size := SIZEOF(activeData);
END_GET
END_PROPERTY

METHOD TryMakeReferenceTo : BOOL
VAR_INPUT
	Target : I_Datatype;
END_VAR
VAR
	pTargetData : POINTER TO TcVnParamsKAZE;
END_VAR
IF NOT IsEquivalentTo(Target) THEN
	RETURN;
END_IF

pTargetData := Target.Address;
activeData REF= pTargetData^;
SetMemberReference();
TryMakeReferenceTo := TRUE;
END_METHOD

PROPERTY PUBLIC Value : REFERENCE TO TcVnParamsKAZE
GET
Value REF= activeData;
END_GET
END_PROPERTY

END_FUNCTION_BLOCK

// ---- Datatypes/Structs/_TcVnParamsORB.TcPOU
{attribute 'linkalways'} 
{attribute 'no_explicit_call' := 'This FB is a CLASS and must be accessed using methods or properties'}
{attribute 'enable_dynamic_creation'}
FUNCTION_BLOCK _TcVnParamsORB EXTENDS StructuredDatatypeBase
VAR
	localData : TcVnParamsORB;
	activeData : REFERENCE TO TcVnParamsORB REF= localData;
    _nMaxPoints : _UDINT(localData.nMaxPoints);
    _fPyramidScale : _REAL(localData.fPyramidScale);
    _nPyramidLevels : _UDINT(localData.nPyramidLevels);
    _nEdgeThreshold : _UDINT(localData.nEdgeThreshold);
    _nFirstLevel : _UDINT(localData.nFirstLevel);
    _nBriefPoints : _UDINT(localData.nBriefPoints);
    _eScoreType : _ETcVnFeatureScoreTypeORB(localData.eScoreType);
    _nPatchSize : _UDINT(localData.nPatchSize);
    _nFastThreshold : _DINT(localData.nFastThreshold);
END_VAR

PROPERTY PUBLIC Address : PVOID
GET
Address := ADR(activeData);
END_GET
END_PROPERTY

METHOD PUBLIC ClearReference
VAR_INPUT
END_VAR
activeData REF= localData;
SetMemberReference();
END_METHOD

METHOD PUBLIC Clone : I_Datatype
VAR
    pClone : POINTER TO _TcVnParamsORB;
END_VAR
pClone := __NEW(_TcVnParamsORB());
pClone^.Value := Value;
Clone := pClone^;
END_METHOD

PROPERTY PUBLIC eScoreType : REFERENCE TO _ETcVnFeatureScoreTypeORB
GET
eScoreType REF= _eScoreType;
END_GET
END_PROPERTY

METHOD FB_init : BOOL
VAR_INPUT
	bInitRetains : BOOL; // if TRUE, the retain variables are initialized (warm start / cold start)
	bInCopyCode : BOOL;  // if TRUE, the instance afterwards gets moved into the copy code (online change)
END_VAR
SetMemberReference();
AddMember('nMaxPoints', _nMaxPoints);
AddMember('fPyramidScale', _fPyramidScale);
AddMember('nPyramidLevels', _nPyramidLevels);
AddMember('nEdgeThreshold', _nEdgeThreshold);
AddMember('nFirstLevel', _nFirstLevel);
AddMember('nBriefPoints', _nBriefPoints);
AddMember('eScoreType', _eScoreType);
AddMember('nPatchSize', _nPatchSize);
AddMember('nFastThreshold', _nFastThreshold);
END_METHOD

PROPERTY PUBLIC fPyramidScale : REFERENCE TO _REAL
GET
fPyramidScale REF= _fPyramidScale;
END_GET
END_PROPERTY

PROPERTY PUBLIC Identifier : T_MAXSTRING
GET
Identifier := 'TcVnParamsORB';
END_GET
END_PROPERTY

METHOD PUBLIC MakeReferenceTo
VAR_INPUT
	ReferenceTarget : REFERENCE TO TcVnParamsORB;
END_VAR
activeData REF= ReferenceTarget;
SetMemberReference();
END_METHOD

PROPERTY PUBLIC nBriefPoints : REFERENCE TO _UDINT
GET
nBriefPoints REF= _nBriefPoints;
END_GET
END_PROPERTY

PROPERTY PUBLIC nEdgeThreshold : REFERENCE TO _UDINT
GET
nEdgeThreshold REF= _nEdgeThreshold;
END_GET
END_PROPERTY

PROPERTY PUBLIC nFastThreshold : REFERENCE TO _DINT
GET
nFastThreshold REF= _nFastThreshold;
END_GET
END_PROPERTY

PROPERTY PUBLIC nFirstLevel : REFERENCE TO _UDINT
GET
nFirstLevel REF= _nFirstLevel;
END_GET
END_PROPERTY

PROPERTY PUBLIC nMaxPoints : REFERENCE TO _UDINT
GET
nMaxPoints REF= _nMaxPoints;
END_GET
END_PROPERTY

PROPERTY PUBLIC nPatchSize : REFERENCE TO _UDINT
GET
nPatchSize REF= _nPatchSize;
END_GET
END_PROPERTY

PROPERTY PUBLIC nPyramidLevels : REFERENCE TO _UDINT
GET
nPyramidLevels REF= _nPyramidLevels;
END_GET
END_PROPERTY

METHOD PROTECTED SetMemberReference
VAR_INPUT
END_VAR
_nMaxPoints.MakeReferenceTo(activeData.nMaxPoints);
_fPyramidScale.MakeReferenceTo(activeData.fPyramidScale);
_nPyramidLevels.MakeReferenceTo(activeData.nPyramidLevels);
_nEdgeThreshold.MakeReferenceTo(activeData.nEdgeThreshold);
_nFirstLevel.MakeReferenceTo(activeData.nFirstLevel);
_nBriefPoints.MakeReferenceTo(activeData.nBriefPoints);
_eScoreType.MakeReferenceTo(activeData.eScoreType);
_nPatchSize.MakeReferenceTo(activeData.nPatchSize);
_nFastThreshold.MakeReferenceTo(activeData.nFastThreshold);
END_METHOD

PROPERTY PUBLIC Size : UDINT
GET
Size := SIZEOF(activeData);
END_GET
END_PROPERTY

METHOD TryMakeReferenceTo : BOOL
VAR_INPUT
	Target : I_Datatype;
END_VAR
VAR
	pTargetData : POINTER TO TcVnParamsORB;
END_VAR
IF NOT IsEquivalentTo(Target) THEN
	RETURN;
END_IF

pTargetData := Target.Address;
activeData REF= pTargetData^;
SetMemberReference();
TryMakeReferenceTo := TRUE;
END_METHOD

PROPERTY PUBLIC Value : REFERENCE TO TcVnParamsORB
GET
Value REF= activeData;
END_GET
END_PROPERTY

END_FUNCTION_BLOCK

// ---- Datatypes/Structs/_TcVnParamsFAST.TcPOU
{attribute 'linkalways'} 
{attribute 'no_explicit_call' := 'This FB is a CLASS and must be accessed using methods or properties'}
{attribute 'enable_dynamic_creation'}
FUNCTION_BLOCK _TcVnParamsFAST EXTENDS StructuredDatatypeBase
VAR
	localData : TcVnParamsFAST;
	activeData : REFERENCE TO TcVnParamsFAST REF= localData;
	_nThreshold : _DINT(localData.nThreshold);
    _bNonMaxSuppression : _BOOL(localData.bNonMaxSuppression);
	_eType : _ETcVnKeypointDetectionTypeFAST(localData.eType);
END_VAR

PROPERTY PUBLIC Address : PVOID
GET
Address := ADR(activeData);
END_GET
END_PROPERTY

PROPERTY PUBLIC bNonMaxSuppression : REFERENCE TO _BOOL
GET
bNonMaxSuppression REF= _bNonMaxSuppression;
END_GET
END_PROPERTY

METHOD PUBLIC ClearReference
VAR_INPUT
END_VAR
activeData REF= localData;
SetMemberReference();
END_METHOD

METHOD PUBLIC Clone : I_Datatype
VAR
    pClone : POINTER TO _TcVnParamsFAST;
END_VAR
pClone := __NEW(_TcVnParamsFAST());
pClone^.Value := Value;
Clone := pClone^;
END_METHOD

PROPERTY PUBLIC eType : REFERENCE TO _ETcVnKeypointDetectionTypeFAST
GET
eType REF= _eType;
END_GET
END_PROPERTY

METHOD FB_init : BOOL
VAR_INPUT
	bInitRetains : BOOL; // if TRUE, the retain variables are initialized (warm start / cold start)
	bInCopyCode : BOOL;  // if TRUE, the instance afterwards gets moved into the copy code (online change)
END_VAR
SetMemberReference();
AddMember('nThreshold',_nThreshold);
AddMember('bNonMaxSuppression',_bNonMaxSuppression );
AddMember('eType',_eType);
END_METHOD

PROPERTY PUBLIC Identifier : T_MAXSTRING
GET
Identifier := 'TcVnParamsFAST';
END_GET
END_PROPERTY

METHOD PUBLIC MakeReferenceTo
VAR_INPUT
	ReferenceTarget : REFERENCE TO TcVnParamsFAST;
END_VAR
activeData REF= ReferenceTarget;
SetMemberReference();
END_METHOD

PROPERTY PUBLIC nThreshold : REFERENCE TO _DINT
GET
nThreshold REF= _nThreshold;
END_GET
END_PROPERTY

METHOD PROTECTED SetMemberReference
VAR_STAT
	// this variable is used for BITADR as this function failes if used on a local variable.
	structure : TcVnPixelFormat;
END_VAR
_nThreshold.MakeReferenceTo(activeData.nThreshold);
_bNonMaxSuppression.MakeReferenceTo(activeData.bNonMaxSuppression);
_eType.MakeReferenceTo(activeData.eType);
END_METHOD

PROPERTY PUBLIC Size : UDINT
GET
Size := SIZEOF(activeData);
END_GET
END_PROPERTY

METHOD TryMakeReferenceTo : BOOL
VAR_INPUT
	Target : I_Datatype;
END_VAR
VAR
	pTargetData : POINTER TO TcVnParamsFAST;
END_VAR
IF NOT IsEquivalentTo(Target) THEN
	RETURN;
END_IF

pTargetData := Target.Address;
activeData REF= pTargetData^;
SetMemberReference();
TryMakeReferenceTo := TRUE;
END_METHOD

PROPERTY PUBLIC Value : REFERENCE TO TcVnParamsFAST
GET
Value REF= activeData;
END_GET
END_PROPERTY

END_FUNCTION_BLOCK

// ---- Datatypes/Structs/_TcVnParamsBlobDetection.TcPOU
{attribute 'linkalways'} 
{attribute 'no_explicit_call' := 'This FB is a CLASS and must be accessed using methods or properties'}
{attribute 'enable_dynamic_creation'}
FUNCTION_BLOCK _TcVnParamsBlobDetection EXTENDS StructuredDatatypeBase
VAR
	localData : TcVnParamsBlobDetection;
	activeData : REFERENCE TO TcVnParamsBlobDetection REF= localData;
    _bFilterByArea         : _BOOL(localdata.bFilterByArea);
    _bFilterByCircularity  : _BOOL(localdata.bFilterByCircularity);
    _bFilterByConvexity    : _BOOL(localdata.bFilterByConvexity);
    _bFilterByEccentricity : _BOOL(localdata.bFilterByEccentricity);
    _bFilterByInertiaRatio : _BOOL(localdata.bFilterByInertiaRatio);
    _fMinArea              : _REAL(localdata.fMinArea);
    _fMaxArea              : _REAL(localdata.fMaxArea);
    _fMinCircularity       : _REAL(localdata.fMinCircularity);
    _fMaxCircularity       : _REAL(localdata.fMaxCircularity);
    _fMinConvexity         : _REAL(localdata.fMinConvexity);
    _fMaxConvexity         : _REAL(localdata.fMaxConvexity);
    _fMinEccentricity      : _REAL(localdata.fMinEccentricity);
    _fMaxEccentricity      : _REAL(localdata.fMaxEccentricity);
    _fMinInertiaRatio      : _REAL(localdata.fMinInertiaRatio);
    _fMaxInertiaRatio      : _REAL(localdata.fMaxInertiaRatio);
    _eThresholdType        : _ETcVnThresholdType(localdata.eThresholdType);
    _fMinThreshold         : _REAL(localdata.fMinThreshold);
    _fMaxThreshold         : _REAL(localdata.fMaxThreshold);
    _fThresholdStep        : _REAL(localdata.fThresholdStep);
    _fMinBlobDistance      : _REAL(localdata.fMinBlobDistance);
    _nMinRepeatability     : _UDINT(localdata.nMinRepeatability);
    _eBlobCombination      : _ETcVnBlobCombination(localdata.eBlobCombination);
END_VAR

PROPERTY PUBLIC Address : PVOID
GET
Address := ADR(activeData);
END_GET
END_PROPERTY

PROPERTY PUBLIC bFilterByArea : REFERENCE TO _BOOL
GET
bFilterByArea REF= _bFilterByArea;
END_GET
END_PROPERTY

PROPERTY PUBLIC bFilterByCircularity : REFERENCE TO _BOOL
GET
bFilterByCircularity REF= _bFilterByCircularity;
END_GET
END_PROPERTY

PROPERTY PUBLIC bFilterByConvexity : REFERENCE TO _BOOL
GET
bFilterByConvexity REF= _bFilterByConvexity;
END_GET
END_PROPERTY

PROPERTY PUBLIC bFilterByEccentricity : REFERENCE TO _BOOL
GET
bFilterByEccentricity REF= _bFilterByEccentricity;
END_GET
END_PROPERTY

PROPERTY PUBLIC bFilterByInertiaRatio : REFERENCE TO _BOOL
GET
bFilterByInertiaRatio REF= _bFilterByInertiaRatio;
END_GET
END_PROPERTY

METHOD PUBLIC ClearReference
VAR_INPUT
END_VAR
activeData REF= localData;
SetMemberReference();
END_METHOD

METHOD PUBLIC Clone : I_Datatype
VAR
    pClone : POINTER TO _TcVnParamsBlobDetection;
END_VAR
pClone := __NEW(_TcVnParamsBlobDetection());
pClone^.Value := Value;
Clone := pClone^;
END_METHOD

PROPERTY PUBLIC eBlobCombination : REFERENCE TO _ETcVnBlobCombination
GET
eBlobCombination REF= _eBlobCombination;
END_GET
END_PROPERTY

PROPERTY PUBLIC eThresholdType : REFERENCE TO _ETcVnThresholdType
GET
eThresholdType REF= _eThresholdType;
END_GET
END_PROPERTY

METHOD FB_init : BOOL
VAR_INPUT
	bInitRetains : BOOL; // if TRUE, the retain variables are initialized (warm start / cold start)
	bInCopyCode : BOOL;  // if TRUE, the instance afterwards gets moved into the copy code (online change)
END_VAR
SetMemberReference();
AddMember('bFilterByArea', _bFilterByArea);
AddMember('bFilterByCircularity', _bFilterByCircularity);
AddMember('bFilterByConvexity', _bFilterByConvexity);
AddMember('bFilterByEccentricity', _bFilterByEccentricity);
AddMember('bFilterByInertiaRatio', _bFilterByInertiaRatio);
AddMember('fMinArea', _fMinArea);
AddMember('fMaxArea', _fMaxArea);
AddMember('fMinCircularity', _fMinCircularity);
AddMember('fMaxCircularity', _fMaxCircularity);
AddMember('fMinConvexity', _fMinConvexity);
AddMember('fMaxConvexity', _fMaxConvexity);
AddMember('fMinEccentricity', _fMinEccentricity);
AddMember('fMaxEccentricity', _fMaxEccentricity);
AddMember('fMinInertiaRatio', _fMinInertiaRatio);
AddMember('fMaxInertiaRatio', _fMaxInertiaRatio);
AddMember('eThresholdType', _eThresholdType);
AddMember('fMinThreshold', _fMinThreshold);
AddMember('fMaxThreshold', _fMaxThreshold);
AddMember('fThresholdStep',  _fThresholdStep);
AddMember('fMinBlobDistance', _fMinBlobDistance);
AddMember('nMinRepeatability', _nMinRepeatability);
AddMember('eBlobCombination', _eBlobCombination);
END_METHOD

PROPERTY PUBLIC fMaxArea : REFERENCE TO _REAL
GET
fMaxArea REF= _fMaxArea;
END_GET
END_PROPERTY

PROPERTY PUBLIC fMaxCircularity : REFERENCE TO _REAL
GET
fMaxCircularity REF= _fMaxCircularity;
END_GET
END_PROPERTY

PROPERTY PUBLIC fMaxConvexity : REFERENCE TO _REAL
GET
fMaxConvexity REF= _fMaxConvexity;
END_GET
END_PROPERTY

PROPERTY PUBLIC fMaxEccentricity : REFERENCE TO _REAL
GET
fMaxEccentricity REF= _fMaxEccentricity;
END_GET
END_PROPERTY

PROPERTY PUBLIC fMaxInertiaRatio : REFERENCE TO _REAL
GET
fMaxInertiaRatio REF= _fMaxInertiaRatio;
END_GET
END_PROPERTY

PROPERTY PUBLIC fMaxThreshold : REFERENCE TO _REAL
GET
fMaxThreshold REF= _fMaxThreshold;
END_GET
END_PROPERTY

PROPERTY PUBLIC fMinArea : REFERENCE TO _REAL
GET
fMinArea REF= _fMinArea;
END_GET
END_PROPERTY

PROPERTY PUBLIC fMinBlobDistance : REFERENCE TO _REAL
GET
fMinBlobDistance REF= _fMinBlobDistance;
END_GET
END_PROPERTY

PROPERTY PUBLIC fMinCircularity : REFERENCE TO _REAL
GET
fMinCircularity REF= _fMinCircularity;
END_GET
END_PROPERTY

PROPERTY PUBLIC fMinConvexity : REFERENCE TO _REAL
GET
fMinConvexity REF= _fMinConvexity;
END_GET
END_PROPERTY

PROPERTY PUBLIC fMinEccentricity : REFERENCE TO _REAL
GET
fMinEccentricity REF= _fMinEccentricity;
END_GET
END_PROPERTY

PROPERTY PUBLIC fMinInertiaRatio : REFERENCE TO _REAL
GET
fMinInertiaRatio REF= _fMinInertiaRatio;
END_GET
END_PROPERTY

PROPERTY PUBLIC fMinThreshold : REFERENCE TO _REAL
GET
fMinThreshold REF= _fMinThreshold;
END_GET
END_PROPERTY

PROPERTY PUBLIC fThresholdStep : REFERENCE TO _REAL
GET
fThresholdStep REF= _fThresholdStep;
END_GET
END_PROPERTY

PROPERTY PUBLIC Identifier : T_MAXSTRING
GET
Identifier := 'TcVnParamsBlobDetection';
END_GET
END_PROPERTY

METHOD PUBLIC MakeReferenceTo
VAR_INPUT
	ReferenceTarget : REFERENCE TO TcVnParamsBlobDetection;
END_VAR
activeData REF= ReferenceTarget;
SetMemberReference();
END_METHOD

PROPERTY PUBLIC nMinRepeatability : REFERENCE TO _UDINT
GET
nMinRepeatability REF= _nMinRepeatability;
END_GET
END_PROPERTY

METHOD PROTECTED SetMemberReference
VAR_INPUT
END_VAR
_bFilterByArea.MakeReferenceTo(activeData.bFilterByArea);
_bFilterByCircularity.MakeReferenceTo(activeData.bFilterByCircularity);
_bFilterByConvexity.MakeReferenceTo(activeData.bFilterByConvexity);
_bFilterByEccentricity.MakeReferenceTo(activeData.bFilterByEccentricity);
_bFilterByInertiaRatio.MakeReferenceTo(activeData.bFilterByInertiaRatio);
_fMinArea.MakeReferenceTo(activeData.fMinArea);
_fMaxArea.MakeReferenceTo(activeData.fMaxArea);
_fMinCircularity.MakeReferenceTo(activeData.fMinCircularity);
_fMaxCircularity.MakeReferenceTo(activeData.fMaxCircularity);
_fMinConvexity.MakeReferenceTo(activeData.fMinConvexity);
_fMaxConvexity.MakeReferenceTo(activeData.fMaxConvexity);
_fMinEccentricity.MakeReferenceTo(activeData.fMinEccentricity);
_fMaxEccentricity.MakeReferenceTo(activeData.fMaxEccentricity);
_fMinInertiaRatio.MakeReferenceTo(activeData.fMinInertiaRatio);
_fMaxInertiaRatio.MakeReferenceTo(activeData.fMaxInertiaRatio);
_eThresholdType.MakeReferenceTo(activeData.eThresholdType);
_fMinThreshold.MakeReferenceTo(activeData.fMinThreshold);
_fMaxThreshold.MakeReferenceTo(activeData.fMaxThreshold);
_fThresholdStep.MakeReferenceTo(activeData.fThresholdStep);
_fMinBlobDistance.MakeReferenceTo(activeData.fMinBlobDistance);
_nMinRepeatability.MakeReferenceTo(activeData.nMinRepeatability);
_eBlobCombination.MakeReferenceTo(activeData.eBlobCombination);
END_METHOD

PROPERTY PUBLIC Size : UDINT
GET
Size := SIZEOF(activeData);
END_GET
END_PROPERTY

METHOD TryMakeReferenceTo : BOOL
VAR_INPUT
	Target : I_Datatype;
END_VAR
VAR
	targetAsStruct : I_StructuredDatatype;
	pTargetData : POINTER TO TcVnParamsBlobDetection;
END_VAR
IF NOT Target.TryResolveAsStructuredDatatype(targetAsStruct) THEN
	RETURN;
END_IF

IF NOT (targetAsStruct.Identifier = Identifier) THEN
	RETURN;
END_IF

pTargetData := Target.Address;
activeData REF= pTargetData^;
SetMemberReference();
TryMakeReferenceTo := TRUE;
END_METHOD

PROPERTY PUBLIC Value : REFERENCE TO TcVnParamsBlobDetection
GET
Value REF= activeData;
END_GET
END_PROPERTY

END_FUNCTION_BLOCK

